// TwinCAT 3 PLC project PLC_MAIN
// ProgramVersion: 3.1.4024.0
// libraries:
//   Tc2_MC2, * (Beckhoff Automation GmbH)
//   Tc2_NC, * (Beckhoff Automation GmbH)
//   Tc2_Standard, * (Beckhoff Automation GmbH)
//   Tc2_System, * (Beckhoff Automation GmbH)
//   Tc2_Utilities, * (Beckhoff Automation GmbH)
//   Tc3_IotBase, * (Beckhoff Automation GmbH)
//   Tc3_JsonXml, * (Beckhoff Automation GmbH)
//   Tc3_Module, * (Beckhoff Automation GmbH)
//   VisuDialogs, * (System)
//   VisuSymbols,3.5.10.0,System
// project tree:
//   DUTs/ E_autoState.TcDUT, E_ECmotorErrorState.TcDUT, E_manualState.TcDUT, E_motorErrorList.TcDUT, E_resetAutoState.TcDUT, E_safetyState.TcDUT, E_teknicMotorMethods.TcDUT, ST_eflexMsgIn.TcDUT, ST_errorRef.TcDUT, ST_ignitionClient.TcDUT
//   / GlobalTextList.TcGTLO, PlcTask.TcTTO, Visualization Manager.TcVMO (not stored), VISU_TASK.TcTTO
//   GVLs/ GVL_devices.TcGVL, GVL_eflex.TcGVL, GVL_ignition.TcGVL, GVL_machine.TcGVL, GVL_persistent.TcGVL
//   POUs/DEVICES/ FB_digitalOut.TcPOU, FB_distSensor2011.TcPOU, FB_estop.TcPOU, FB_ltBar.TcPOU, FB_ltCurtains.TcPOU, FB_pushBtnNC.TcPOU, FB_pushBtnNO.TcPOU, FB_table.TcPOU, FB_teknicMotorEC.TcPOU
//   POUs/FUNCTIONS/ FB_homeToTorque.TcPOU, FB_homeToSensorCustom.TcPOU, FB_ignitionClientHandler.TcPOU, FB_moveToTorque.TcPOU, FB_MultiMotorController.TcPOU, F_checkCoupledMovement.TcPOU, F_checkMoveFinish.TcPOU, F_recordErrorData.TcPOU
//   POUs/ICONS/ Icons.TcIPO (not stored)
//   POUs/LISTS/ actionSelectList.TcTLO
//   POUs/PROGRAMS/ auto.TcPOU, eflex.TcPOU, errorHandling.TcPOU, MAIN.TcPOU, multiControl.TcPOU, manual.TcPOU, motorsInit.TcPOU, tempEflex.TcPOU, updateMotors.TcPOU
//   VISUs/VISUs/Auto Screens/ baseInSkiOutScreen.TcVIS, continueAutoScreen.TcVIS, eflexScreen.TcVIS, loadSpaScreen.TcVIS, machineHomingScreen.TcVIS, studsInScreen.TcVIS, tempEflexScreen.TcVIS, unloadSpaScreen.TcVIS
//   VISUs/VISUs/multiControlScreens/ parametersScreen.TcVIS, multiControlHelp.TcVIS, multiControlScreen.TcVIS, machineMapScreen.TcVIS, motorControlScreen.TcVIS
//   VISUs/VISUs/ errorScreen.TcVIS, mainScreen.TcVIS, manualBypassedScreen.TcVIS, manualScreen.TcVIS, safetyDisableWarning.TcVIS, safetyResetScreen.TcVIS, settingsScreen.TcVIS
// real-time tasks:
//   TASK PlcTask: cycle T#5ms, priority 10, ADS port 350
//   TASK VISU_TASK: cycle T#100000us, priority 12, ADS port 351
// motion (NC):
//   TASK NC-Task 1 SAF: cycle T#1ms, priority 4, ADS port 501
//   TASK NC-Task 1 SVB: cycle T#1ms, priority 6, ADS port 511
//   AXIS LFTROTATION (id 2)
//     General: UnitName=°
//     Dynamic: AccelerationMaximum=55, DecelerationMaximum=55, Acceleration=50, Deceleration=50
//     Velo: RefSearch=3, RefSync=3, SlowManual=5, FastManual=9, Maximum=10
//     OtherSettings: AllowMotionCmdToSlave=true
//     encoder EncType=19
//       EncPara: ScaleFactorNumerator=7.028e-05, MaxCount=#xffffffff
//         SoftEndMinControl: Enable=true, Range=-290
//         SoftEndMaxControl: Enable=true, Range=-65.5
//     drive DrvType=16
//       DrvPara: MaxCount=#xffffffff, DriveControlDWord=#x00020100
//         Analog: VeloReferenz=8, TorqueSetpointScale=10, ScaleFactorActTorque=0.1
//         TimeComp: TaskDelayCycles=1
//     controller CtrType=1
//       CtrPara: PriorControlFactor=1
//         Observer: BandWidth=20
//   AXIS LFTCLAMP (id 1)
//     Dynamic: AccelerationMaximum=105, DecelerationMaximum=105, Acceleration=100, Deceleration=100
//     Velo: RefSearch=20, RefSync=20, SlowManual=20, FastManual=30, Maximum=35
//     OtherSettings: AllowMotionCmdToSlave=true
//     encoder EncType=19
//       EncPara: ScaleFactorNumerator=4.8672e-05, MaxCount=#xffffffff
//         SoftEndMinControl: Enable=true, Range=-260
//         SoftEndMaxControl: Enable=true
//     drive DrvType=16
//       DrvPara: MaxCount=#xffffffff, DriveControlDWord=#x00020100
//         Analog: VeloReferenz=20, TorqueSetpointScale=10, ScaleFactorActTorque=0.1
//         TimeComp: TaskDelayCycles=1
//     controller CtrType=1
//       CtrPara: PriorControlFactor=1
//         Observer: BandWidth=20
//   AXIS Column1 (id 4)
//     Dynamic: AccelerationMaximum=201, DecelerationMaximum=201, Acceleration=200, Deceleration=200
//     Velo: RefSearch=10, RefSync=10, SlowManual=5, FastManual=10, Maximum=15
//     OtherSettings: AllowMotionCmdToSlave=true
//     encoder EncType=19
//       EncPara: ScaleFactorNumerator=9.75e-05, ScaleFactorDenominator=10, MaxCount=#xffffffff
//         SoftEndMinControl: Enable=true, Range=-622
//         SoftEndMaxControl: Range=0.1
//     drive DrvType=16
//       DrvPara: MaxCount=#xffffffff, DriveControlDWord=#x00020100
//         Analog: VeloReferenz=10, TorqueSetpointScale=10, ScaleFactorActTorque=0.1
//         TimeComp: TaskDelayCycles=1
//     controller CtrType=1
//       CtrPara: PriorControlFactor=1
//         Observer: BandWidth=20
//   AXIS LFTWIDTH (id 5)
//     Dynamic: AccelerationMaximum=55, DecelerationMaximum=55, Acceleration=50, Deceleration=50
//     Velo: RefSearch=10, RefSync=10, SlowManual=10, FastManual=20, Maximum=25
//     OtherSettings: AllowMotionCmdToSlave=true
//     encoder EncType=19
//       EncPara: ScaleFactorNumerator=9.7263e-05, MaxCount=#xffffffff
//         SoftEndMinControl: Enable=true
//         SoftEndMaxControl: Enable=true, Range=430
//     drive DrvType=16
//       DrvPara: MaxCount=#xffffffff, DriveControlDWord=#x00020100
//         Analog: VeloReferenz=20, TorqueSetpointScale=10, ScaleFactorActTorque=0.1
//         TimeComp: TaskDelayCycles=1
//     controller CtrType=1
//       CtrPara: PriorControlFactor=1
//         Observer: BandWidth=20
//   AXIS RHTWIDTH (id 6)
//     Dynamic: AccelerationMaximum=55, DecelerationMaximum=55, Acceleration=50, Deceleration=50
//     Velo: RefSearch=10, RefSync=10, SlowManual=20, FastManual=20, Maximum=25
//     OtherSettings: AllowMotionCmdToSlave=true
//     encoder EncType=19
//       EncPara: ScaleFactorNumerator=9.7263e-05, MaxCount=#xffffffff
//         SoftEndMinControl: Enable=true
//         SoftEndMaxControl: Enable=true, Range=430
//     drive DrvType=16
//       DrvPara: MaxCount=#xffffffff, DriveControlDWord=#x00020100
//         Analog: VeloReferenz=20, TorqueSetpointScale=10, ScaleFactorActTorque=0.1
//         TimeComp: TaskDelayCycles=1
//     controller CtrType=1
//       CtrPara: PriorControlFactor=1
//         Observer: BandWidth=20
//   AXIS Column2 (id 7)
//     Dynamic: AccelerationMaximum=201, DecelerationMaximum=201, Acceleration=200, Deceleration=200
//     Velo: RefSearch=10, RefSync=10, Maximum=15
//     OtherSettings: AllowMotionCmdToSlave=true
//     encoder EncType=19
//       EncPara: ScaleFactorNumerator=9.75e-05, ScaleFactorDenominator=10, MaxCount=#xffffffff
//         SoftEndMinControl: Enable=true, Range=-622
//         SoftEndMaxControl: Enable=true
//     drive DrvType=16
//       DrvPara: MaxCount=#xffffffff, DriveControlDWord=#x00020100
//         Analog: VeloReferenz=10, TorqueSetpointScale=10, ScaleFactorActTorque=0.1
//         TimeComp: TaskDelayCycles=1
//     controller CtrType=1
//       CtrPara: PriorControlFactor=1
//         Observer: BandWidth=20
//   AXIS Column3 (id 8)
//     Dynamic: AccelerationMaximum=201, DecelerationMaximum=201, Acceleration=200, Deceleration=200
//     Velo: RefSearch=10, RefSync=10, Maximum=15
//     OtherSettings: AllowMotionCmdToSlave=true
//     encoder EncType=19
//       EncPara: ScaleFactorNumerator=9.75e-05, ScaleFactorDenominator=10, MaxCount=#xffffffff
//         SoftEndMinControl: Enable=true, Range=-622
//         SoftEndMaxControl: Range=0.1
//     drive DrvType=16
//       DrvPara: MaxCount=#xffffffff, DriveControlDWord=#x00020100
//         Analog: VeloReferenz=10, TorqueSetpointScale=10, ScaleFactorActTorque=0.1
//         TimeComp: TaskDelayCycles=1
//     controller CtrType=1
//       CtrPara: PriorControlFactor=1
//         Observer: BandWidth=20
//   AXIS RHTCLAMP (id 9)
//     Dynamic: AccelerationMaximum=105, DecelerationMaximum=105, Acceleration=100, Deceleration=100
//     Velo: RefSearch=20, RefSync=20, SlowManual=20, FastManual=30, Maximum=35
//     OtherSettings: AllowMotionCmdToSlave=true
//     encoder EncType=19
//       EncPara: ScaleFactorNumerator=4.8672e-05, MaxCount=#xffffffff
//         SoftEndMinControl: Enable=true
//         SoftEndMaxControl: Enable=true, Range=260
//     drive DrvType=16
//       DrvPara: MaxCount=#xffffffff, DriveControlDWord=#x00020100
//         Analog: VeloReferenz=20, TorqueSetpointScale=10, ScaleFactorActTorque=0.1
//         TimeComp: TaskDelayCycles=1
//     controller CtrType=1
//       CtrPara: PriorControlFactor=1
//         Observer: BandWidth=20
//   AXIS RHTROTATION (id 10)
//     General: UnitName=°
//     Dynamic: AccelerationMaximum=55, DecelerationMaximum=55, Acceleration=50, Deceleration=50
//     Velo: RefSearch=3, RefSync=3, Maximum=10
//     OtherSettings: AllowMotionCmdToSlave=true
//     encoder EncType=19
//       EncPara: ScaleFactorNumerator=7.028e-05, MaxCount=#xffffffff
//         SoftEndMinControl: Enable=true, Range=67
//         SoftEndMaxControl: Enable=true, Range=290
//     drive DrvType=16
//       DrvPara: MaxCount=#xffffffff, DriveControlDWord=#x00020100
//         Analog: VeloReferenz=8, TorqueSetpointScale=10, ScaleFactorActTorque=0.1
//         TimeComp: TaskDelayCycles=1
//     controller CtrType=1
//       CtrPara: PriorControlFactor=1
//         Observer: BandWidth=20
//   AXIS Column0 (id 11)
//     Dynamic: AccelerationMaximum=201, DecelerationMaximum=201, Acceleration=200, Deceleration=200
//     Velo: RefSearch=10, RefSync=10, SlowManual=10, FastManual=10, Maximum=15
//     OtherSettings: AllowMotionCmdToSlave=true
//     encoder EncType=19
//       EncPara: ScaleFactorNumerator=9.75e-05, ScaleFactorDenominator=10, MaxCount=#xffffffff
//         SoftEndMinControl: Enable=true, Range=-622
//         SoftEndMaxControl: Enable=true
//     drive DrvType=16
//       DrvPara: MaxCount=#xffffffff, DriveControlDWord=#x00020100
//         Analog: VeloReferenz=10, TorqueSetpointScale=10, ScaleFactorActTorque=0.1
//         TimeComp: TaskDelayCycles=1
//     controller CtrType=1
//       CtrPara: PriorControlFactor=1
//         Observer: BandWidth=20
// I/O:
//   DEVICE Device 1 (EtherCAT), AmsNetId 5.151.65.180.2.1
//     Term 10 (EK1200) [EK1200-5000 EtherCAT Power supply (2A E-Bus)]
//       Term 11 (EL1008) [EL1008 8Ch. Dig. Input 24V, 3ms]
//       Term 12 (EL2008) [EL2008 8Ch. Dig. Output 24V, 0.5A]
//       Term 13 (EL2008) [EL2008 8Ch. Dig. Output 24V, 0.5A]
//       Term 14 (EL2904) [EL2904, 4 Ch. Safety Output 24V, 0.5A, TwinSAFE]
//         modules: Module 1 (FSOES), Module 2 (DO)
//       Term 15 (EL3024) [EL3024 4Ch. Ana. Input 4-20mA DIFF]
//       Term 16 (EL3024) [EL3024 4Ch. Ana. Input 4-20mA DIFF]
//       Term 17 (EL1918) [EL1918, 8Ch. Safety Input 24V, TwinSAFE]
//         modules: Module 2 (FSLOGIC)
//       Term 18 (EK1110) [EK1110 EtherCAT extension]
//     Drive 19 (ClearPath EtherCAT Integrated ServoMotor) [ClearPath EC (CoE Rev 2)]
//     Drive 20 (ClearPath EtherCAT Integrated ServoMotor) [ClearPath EC (CoE Rev 2)]
//     Drive 21 (ClearPath EtherCAT Integrated ServoMotor) [ClearPath EC (CoE Rev 2)]
//     Drive 22 (ClearPath EtherCAT Integrated ServoMotor) [ClearPath EC (CoE Rev 2)]
//     Drive 23 (ClearPath EtherCAT Integrated ServoMotor) [ClearPath EC (CoE Rev 2)]
//     Drive 24 (ClearPath EtherCAT Integrated ServoMotor) [ClearPath EC (CoE Rev 2)]
//     Drive 25 (ClearPath EtherCAT Integrated ServoMotor) [ClearPath EC (CoE Rev 2)]
//     Drive 26 (ClearPath EtherCAT Integrated ServoMotor) [ClearPath EC (CoE Rev 2)]
//     Drive 37 (ClearPath EtherCAT Integrated ServoMotor) [ClearPath EC (CoE Rev 2)]
//     Drive 28 (ClearPath EtherCAT Integrated ServoMotor) [ClearPath EC (CoE Rev 2)]
// variable links:
//   PLC_MAIN/PLC_MAIN Instance <-> Device 1 (EtherCAT)/Term 10 (EK1200)/Term 11 (EL1008)
//     PlcTask Inputs/GVL_devices.fbColumn0Motor.bHomeSensor <-> Channel 6/Input
//     PlcTask Inputs/GVL_devices.fbColumn2Motor.bHomeSensor <-> Channel 5/Input
//     PlcTask Inputs/GVL_devices.fbLftWidthMotor.bClampSensor <-> Channel 1/Input
//     PlcTask Inputs/GVL_devices.fbLftWidthMotor.bHomeSensor <-> Channel 4/Input
//     PlcTask Inputs/GVL_devices.fbRhtWidthMotor.bClampSensor <-> Channel 2/Input
//     PlcTask Inputs/GVL_devices.fbRhtWidthMotor.bHomeSensor <-> Channel 3/Input
//     PlcTask Inputs/GVL_devices.fbTable.bLoadedSensor <-> Channel 7/Input
//   PLC_MAIN/PLC_MAIN Instance <-> Device 1 (EtherCAT)/Term 10 (EK1200)/Term 12 (EL2008)
//     PlcTask Outputs/GVL_devices.fbLftClampMotor.bBrake <-> Channel 7/Output
//     PlcTask Outputs/GVL_devices.fbLftRotationMotor.bBrake <-> Channel 4/Output
//     PlcTask Outputs/GVL_devices.fbLtBars.bGreenLight <-> Channel 1/Output
//     PlcTask Outputs/GVL_devices.fbLtBars.bRedLight <-> Channel 3/Output
//     PlcTask Outputs/GVL_devices.fbLtBars.bYellowLight <-> Channel 2/Output
//     PlcTask Outputs/GVL_devices.fbRhtClampMotor.bBrake <-> Channel 6/Output
//     PlcTask Outputs/GVL_devices.fbRhtRotationMotor.bBrake <-> Channel 5/Output
//   PLC_MAIN/PLC_MAIN Instance <-> Device 1 (EtherCAT)/Term 10 (EK1200)/Term 13 (EL2008)
//     PlcTask Outputs/GVL_devices.fbTable.bTableBlackWire <-> Channel 5/Output
//     PlcTask Outputs/GVL_devices.fbTable.bTableBlueWire <-> Channel 6/Output
//     PlcTask Outputs/GVL_devices.fbTable.bTableGreenWire <-> Channel 4/Output
//   PLC_MAIN/PLC_MAIN Instance <-> Device 1 (EtherCAT)/Term 10 (EK1200)/Term 16 (EL3024)
//     PlcTask Inputs/GVL_devices.fbTable.tableDistSens.nSensor <-> AI Standard Channel 1/Value
//   PLC_MAIN/PLC_MAIN Instance <-> Device 1 (EtherCAT)/Term 10 (EK1200)/Term 17 (EL1918)
//     PlcTask Inputs/GVL_devices.fbEstop.bEstopFbError <-> StandardInputs/Standard Out Var 18
//     PlcTask Inputs/GVL_devices.fbEstop.bEstopSigOk <-> StandardInputs/Standard Out Var 19
//     PlcTask Inputs/GVL_devices.fbEstop.nEstopFbState <-> Function Block Info Data/TwinSafeGroup1.Network1.FBEstop1 Info Data/State
//     PlcTask Inputs/GVL_devices.fbLtCurtains.bCurtainsMuted <-> StandardInputs/Standard Out Var 17
//     PlcTask Inputs/GVL_devices.fbLtCurtains.bLftCurtainFbError <-> StandardInputs/Standard Out Var 11
//     PlcTask Inputs/GVL_devices.fbLtCurtains.bLftCurtainSigOk <-> StandardInputs/Standard Out Var 12
//     PlcTask Inputs/GVL_devices.fbLtCurtains.bRhtCurtainFbError <-> StandardInputs/Standard Out Var 14
//     PlcTask Inputs/GVL_devices.fbLtCurtains.bRhtCurtainSigOk <-> StandardInputs/Standard Out Var 15
//     PlcTask Inputs/GVL_devices.fbLtCurtains.nLftCurtainFbState <-> Function Block Info Data/TwinSafeGroup1.Network1.FBMon1 Info Data/State
//     PlcTask Inputs/GVL_devices.fbLtCurtains.nRhtCurtainFbState <-> Function Block Info Data/TwinSafeGroup1.Network1.FBMon2 Info Data/State
//     PlcTask Inputs/GVL_machine.bComErr <-> StandardInputs/Standard Out Var 8
//     PlcTask Inputs/GVL_machine.bFbErr <-> StandardInputs/Standard Out Var 20
//     PlcTask Inputs/GVL_machine.bFbRun <-> StandardInputs/Standard Out Var 9
//     PlcTask Inputs/GVL_machine.bInRun <-> StandardInputs/Standard Out Var 10
//     PlcTask Inputs/GVL_machine.bOtherErr <-> StandardInputs/Standard Out Var 13
//     PlcTask Inputs/GVL_machine.bSafetyOk <-> StandardInputs/Standard Out Var 16
//     PlcTask Outputs/GVL_devices.fbEstop.bResetEstopFb <-> StandardOutputs/Standard In Var 4
//     PlcTask Outputs/GVL_devices.fbLtCurtains.bMuteCurtains <-> StandardOutputs/Standard In Var 3
//     PlcTask Outputs/GVL_devices.fbLtCurtains.bResetLftCurtainFb <-> StandardOutputs/Standard In Var 5
//     PlcTask Outputs/GVL_devices.fbLtCurtains.bResetRhtCurtainFb <-> StandardOutputs/Standard In Var 6
//     PlcTask Outputs/GVL_machine.bRunSafety <-> StandardOutputs/Standard In Var 2
//     PlcTask Outputs/GVL_machine.bSafetyBypass <-> StandardOutputs/Standard In Var 7
//     PlcTask Outputs/GVL_machine.bSafetyErrorAck <-> StandardOutputs/Standard In Var 1
//   PLC_MAIN/PLC_MAIN Instance <-> NC-Task 1 SAF/Axes/Column0
//     PlcTask Inputs/GVL_devices.fbColumn0Motor.fbMotor.NcToPlc <-> Outputs/ToPlc
//     PlcTask Outputs/GVL_devices.fbColumn0Motor.fbMotor.PlcToNc <-> Inputs/FromPlc
//   PLC_MAIN/PLC_MAIN Instance <-> NC-Task 1 SAF/Axes/Column1
//     PlcTask Inputs/GVL_devices.fbColumn1Motor.fbMotor.NcToPlc <-> Outputs/ToPlc
//     PlcTask Outputs/GVL_devices.fbColumn1Motor.fbMotor.PlcToNc <-> Inputs/FromPlc
//   PLC_MAIN/PLC_MAIN Instance <-> NC-Task 1 SAF/Axes/Column2
//     PlcTask Inputs/GVL_devices.fbColumn2Motor.fbMotor.NcToPlc <-> Outputs/ToPlc
//     PlcTask Outputs/GVL_devices.fbColumn2Motor.fbMotor.PlcToNc <-> Inputs/FromPlc
//   PLC_MAIN/PLC_MAIN Instance <-> NC-Task 1 SAF/Axes/Column3
//     PlcTask Inputs/GVL_devices.fbColumn3Motor.fbMotor.NcToPlc <-> Outputs/ToPlc
//     PlcTask Outputs/GVL_devices.fbColumn3Motor.fbMotor.PlcToNc <-> Inputs/FromPlc
//   PLC_MAIN/PLC_MAIN Instance <-> NC-Task 1 SAF/Axes/LFTCLAMP
//     PlcTask Inputs/GVL_devices.fbLftClampMotor.fbMotor.NcToPlc <-> Outputs/ToPlc
//     PlcTask Outputs/GVL_devices.fbLftClampMotor.fbMotor.PlcToNc <-> Inputs/FromPlc
//   PLC_MAIN/PLC_MAIN Instance <-> NC-Task 1 SAF/Axes/LFTROTATION
//     PlcTask Inputs/GVL_devices.fbLftRotationMotor.fbMotor.NcToPlc <-> Outputs/ToPlc
//     PlcTask Outputs/GVL_devices.fbLftRotationMotor.fbMotor.PlcToNc <-> Inputs/FromPlc
//   PLC_MAIN/PLC_MAIN Instance <-> NC-Task 1 SAF/Axes/LFTWIDTH
//     PlcTask Inputs/GVL_devices.fbLftWidthMotor.fbMotor.NcToPlc <-> Outputs/ToPlc
//     PlcTask Outputs/GVL_devices.fbLftWidthMotor.fbMotor.PlcToNc <-> Inputs/FromPlc
//   PLC_MAIN/PLC_MAIN Instance <-> NC-Task 1 SAF/Axes/RHTCLAMP
//     PlcTask Inputs/GVL_devices.fbRhtClampMotor.fbMotor.NcToPlc <-> Outputs/ToPlc
//     PlcTask Outputs/GVL_devices.fbRhtClampMotor.fbMotor.PlcToNc <-> Inputs/FromPlc
//   PLC_MAIN/PLC_MAIN Instance <-> NC-Task 1 SAF/Axes/RHTROTATION
//     PlcTask Inputs/GVL_devices.fbRhtRotationMotor.fbMotor.NcToPlc <-> Outputs/ToPlc
//     PlcTask Outputs/GVL_devices.fbRhtRotationMotor.fbMotor.PlcToNc <-> Inputs/FromPlc
//   PLC_MAIN/PLC_MAIN Instance <-> NC-Task 1 SAF/Axes/RHTWIDTH
//     PlcTask Inputs/GVL_devices.fbRhtWidthMotor.fbMotor.NcToPlc <-> Outputs/ToPlc
//     PlcTask Outputs/GVL_devices.fbRhtWidthMotor.fbMotor.PlcToNc <-> Inputs/FromPlc
//   Axes/LFTROTATION <-> Device 1 (EtherCAT)/Drive 19 (ClearPath EtherCAT Integrated ServoMotor)
//     Drive/Inputs/In/nDataIn1 <-> TxPDO 1/Following Error Actual Value
//     Drive/Inputs/In/nDataIn3[0] <-> TxPDO 1/Torque Actual Value
//     Drive/Inputs/In/nState1 <-> TxPDO 1/Statusword
//     Drive/Inputs/In/nState2 <-> TxPDO 1/Statusword @bit 8
//     Drive/Inputs/In/nState4 @bit 1 <-> WcState/InputToggle
//     Drive/Inputs/In/nState4 <-> WcState/WcState
//     Drive/Inputs/In/nState5 <-> TxPDO 1/Modes of Operation Display
//     Drive/Outputs/Out/nCtrl1 <-> RxPDO 1/Controlword
//     Drive/Outputs/Out/nCtrl2 <-> RxPDO 1/Controlword @bit 8
//     Drive/Outputs/Out/nCtrl5 <-> RxPDO 1/Modes of Operation
//     Drive/Outputs/Out/nDataOut1 <-> RxPDO 1/Target Position
//     Drive/Outputs/Out/nDataOut2 <-> RxPDO 1/Target Velocity
//     Drive/Outputs/Out/nDataOut4[0] <-> RxPDO 1/Target Torque
//     Enc/Inputs/In/nDataIn1 <-> TxPDO 1/Position Actual Value
//     Enc/Inputs/In/nDataIn7 <-> TxPDO 1/Velocity Actual Value
//     Enc/Inputs/In/nState4 @bit 1 <-> WcState/InputToggle
//     Enc/Inputs/In/nState4 <-> WcState/WcState
//   (this object) <-> Device 1 (EtherCAT)/Drive 20 (ClearPath EtherCAT Integrated ServoMotor)
//     Drive/Inputs/In/nDataIn1 <-> TxPDO 1/Following Error Actual Value
//     Drive/Inputs/In/nDataIn3[0] <-> TxPDO 1/Torque Actual Value
//     Drive/Inputs/In/nState1 <-> TxPDO 1/Statusword
//     Drive/Inputs/In/nState2 <-> TxPDO 1/Statusword @bit 8
//     Drive/Inputs/In/nState4 @bit 1 <-> WcState/InputToggle
//     Drive/Inputs/In/nState4 <-> WcState/WcState
//     Drive/Inputs/In/nState5 <-> TxPDO 1/Modes of Operation Display
//     Drive/Outputs/Out/nCtrl1 <-> RxPDO 1/Controlword
//     Drive/Outputs/Out/nCtrl2 <-> RxPDO 1/Controlword @bit 8
//     Drive/Outputs/Out/nCtrl5 <-> RxPDO 1/Modes of Operation
//     Drive/Outputs/Out/nDataOut1 <-> RxPDO 1/Target Position
//     Drive/Outputs/Out/nDataOut2 <-> RxPDO 1/Target Velocity
//     Drive/Outputs/Out/nDataOut4[0] <-> RxPDO 1/Target Torque
//     Enc/Inputs/In/nDataIn1 <-> TxPDO 1/Position Actual Value
//     Enc/Inputs/In/nDataIn7 <-> TxPDO 1/Velocity Actual Value
//     Enc/Inputs/In/nState4 @bit 1 <-> WcState/InputToggle
//     Enc/Inputs/In/nState4 <-> WcState/WcState
//   (this object) <-> Device 1 (EtherCAT)/Drive 22 (ClearPath EtherCAT Integrated ServoMotor)
//     Drive/Inputs/In/nDataIn1 <-> TxPDO 1/Following Error Actual Value
//     Drive/Inputs/In/nDataIn3[0] <-> TxPDO 1/Torque Actual Value
//     Drive/Inputs/In/nState1 <-> TxPDO 1/Statusword
//     Drive/Inputs/In/nState2 <-> TxPDO 1/Statusword @bit 8
//     Drive/Inputs/In/nState4 @bit 1 <-> WcState/InputToggle
//     Drive/Inputs/In/nState4 <-> WcState/WcState
//     Drive/Inputs/In/nState5 <-> TxPDO 1/Modes of Operation Display
//     Drive/Outputs/Out/nCtrl1 <-> RxPDO 1/Controlword
//     Drive/Outputs/Out/nCtrl2 <-> RxPDO 1/Controlword @bit 8
//     Drive/Outputs/Out/nCtrl5 <-> RxPDO 1/Modes of Operation
//     Drive/Outputs/Out/nDataOut1 <-> RxPDO 1/Target Position
//     Drive/Outputs/Out/nDataOut2 <-> RxPDO 1/Target Velocity
//     Drive/Outputs/Out/nDataOut4[0] <-> RxPDO 1/Target Torque
//     Enc/Inputs/In/nDataIn1 <-> TxPDO 1/Position Actual Value
//     Enc/Inputs/In/nDataIn7 <-> TxPDO 1/Velocity Actual Value
//     Enc/Inputs/In/nState4 @bit 1 <-> WcState/InputToggle
//     Enc/Inputs/In/nState4 <-> WcState/WcState
//   (this object) <-> Device 1 (EtherCAT)/Drive 23 (ClearPath EtherCAT Integrated ServoMotor)
//     Drive/Inputs/In/nDataIn1 <-> TxPDO 1/Following Error Actual Value
//     Drive/Inputs/In/nDataIn3[0] <-> TxPDO 1/Torque Actual Value
//     Drive/Inputs/In/nState1 <-> TxPDO 1/Statusword
//     Drive/Inputs/In/nState2 <-> TxPDO 1/Statusword @bit 8
//     Drive/Inputs/In/nState4 @bit 1 <-> WcState/InputToggle
//     Drive/Inputs/In/nState4 <-> WcState/WcState
//     Drive/Inputs/In/nState5 <-> TxPDO 1/Modes of Operation Display
//     Drive/Outputs/Out/nCtrl1 <-> RxPDO 1/Controlword
//     Drive/Outputs/Out/nCtrl2 <-> RxPDO 1/Controlword @bit 8
//     Drive/Outputs/Out/nCtrl5 <-> RxPDO 1/Modes of Operation
//     Drive/Outputs/Out/nDataOut1 <-> RxPDO 1/Target Position
//     Drive/Outputs/Out/nDataOut2 <-> RxPDO 1/Target Velocity
//     Drive/Outputs/Out/nDataOut4[0] <-> RxPDO 1/Target Torque
//     Enc/Inputs/In/nDataIn1 <-> TxPDO 1/Position Actual Value
//     Enc/Inputs/In/nDataIn7 <-> TxPDO 1/Velocity Actual Value
//     Enc/Inputs/In/nState4 @bit 1 <-> WcState/InputToggle
//     Enc/Inputs/In/nState4 <-> WcState/WcState
//   (this object) <-> Device 1 (EtherCAT)/Drive 24 (ClearPath EtherCAT Integrated ServoMotor)
//     Drive/Inputs/In/nDataIn1 <-> TxPDO 1/Following Error Actual Value
//     Drive/Inputs/In/nDataIn3[0] <-> TxPDO 1/Torque Actual Value
//     Drive/Inputs/In/nState1 <-> TxPDO 1/Statusword
//     Drive/Inputs/In/nState2 <-> TxPDO 1/Statusword @bit 8
//     Drive/Inputs/In/nState4 @bit 1 <-> WcState/InputToggle
//     Drive/Inputs/In/nState4 <-> WcState/WcState
//     Drive/Inputs/In/nState5 <-> TxPDO 1/Modes of Operation Display
//     Drive/Outputs/Out/nCtrl1 <-> RxPDO 1/Controlword
//     Drive/Outputs/Out/nCtrl2 <-> RxPDO 1/Controlword @bit 8
//     Drive/Outputs/Out/nCtrl5 <-> RxPDO 1/Modes of Operation
//     Drive/Outputs/Out/nDataOut1 <-> RxPDO 1/Target Position
//     Drive/Outputs/Out/nDataOut2 <-> RxPDO 1/Target Velocity
//     Drive/Outputs/Out/nDataOut4[0] <-> RxPDO 1/Target Torque
//     Enc/Inputs/In/nDataIn1 <-> TxPDO 1/Position Actual Value
//     Enc/Inputs/In/nDataIn7 <-> TxPDO 1/Velocity Actual Value
//     Enc/Inputs/In/nState4 @bit 1 <-> WcState/InputToggle
//     Enc/Inputs/In/nState4 <-> WcState/WcState
//   (this object) <-> Device 1 (EtherCAT)/Drive 25 (ClearPath EtherCAT Integrated ServoMotor)
//     Drive/Inputs/In/nDataIn1 <-> TxPDO 1/Following Error Actual Value
//     Drive/Inputs/In/nDataIn3[0] <-> TxPDO 1/Torque Actual Value
//     Drive/Inputs/In/nState1 <-> TxPDO 1/Statusword
//     Drive/Inputs/In/nState2 <-> TxPDO 1/Statusword @bit 8
//     Drive/Inputs/In/nState4 @bit 1 <-> WcState/InputToggle
//     Drive/Inputs/In/nState4 <-> WcState/WcState
//     Drive/Inputs/In/nState5 <-> TxPDO 1/Modes of Operation Display
//     Drive/Outputs/Out/nCtrl1 <-> RxPDO 1/Controlword
//     Drive/Outputs/Out/nCtrl2 <-> RxPDO 1/Controlword @bit 8
//     Drive/Outputs/Out/nCtrl5 <-> RxPDO 1/Modes of Operation
//     Drive/Outputs/Out/nDataOut1 <-> RxPDO 1/Target Position
//     Drive/Outputs/Out/nDataOut2 <-> RxPDO 1/Target Velocity
//     Drive/Outputs/Out/nDataOut4[0] <-> RxPDO 1/Target Torque
//     Enc/Inputs/In/nDataIn1 <-> TxPDO 1/Position Actual Value
//     Enc/Inputs/In/nDataIn7 <-> TxPDO 1/Velocity Actual Value
//     Enc/Inputs/In/nState4 @bit 1 <-> WcState/InputToggle
//     Enc/Inputs/In/nState4 <-> WcState/WcState
//   (this object) <-> Device 1 (EtherCAT)/Drive 26 (ClearPath EtherCAT Integrated ServoMotor)
//     Drive/Inputs/In/nDataIn1 <-> TxPDO 1/Following Error Actual Value
//     Drive/Inputs/In/nDataIn3[0] <-> TxPDO 1/Torque Actual Value
//     Drive/Inputs/In/nState1 <-> TxPDO 1/Statusword
//     Drive/Inputs/In/nState2 <-> TxPDO 1/Statusword @bit 8
//     Drive/Inputs/In/nState4 @bit 1 <-> WcState/InputToggle
//     Drive/Inputs/In/nState4 <-> WcState/WcState
//     Drive/Inputs/In/nState5 <-> TxPDO 1/Modes of Operation Display
//     Drive/Outputs/Out/nCtrl1 <-> RxPDO 1/Controlword
//     Drive/Outputs/Out/nCtrl2 <-> RxPDO 1/Controlword @bit 8
//     Drive/Outputs/Out/nCtrl5 <-> RxPDO 1/Modes of Operation
//     Drive/Outputs/Out/nDataOut1 <-> RxPDO 1/Target Position
//     Drive/Outputs/Out/nDataOut2 <-> RxPDO 1/Target Velocity
//     Drive/Outputs/Out/nDataOut4[0] <-> RxPDO 1/Target Torque
//     Enc/Inputs/In/nDataIn1 <-> TxPDO 1/Position Actual Value
//     Enc/Inputs/In/nDataIn7 <-> TxPDO 1/Velocity Actual Value
//     Enc/Inputs/In/nState4 @bit 1 <-> WcState/InputToggle
//     Enc/Inputs/In/nState4 <-> WcState/WcState
//   (this object) <-> Device 1 (EtherCAT)/Drive 37 (ClearPath EtherCAT Integrated ServoMotor)
//     Drive/Inputs/In/nDataIn1 <-> TxPDO 1/Following Error Actual Value
//     Drive/Inputs/In/nDataIn3[0] <-> TxPDO 1/Torque Actual Value
//     Drive/Inputs/In/nState1 <-> TxPDO 1/Statusword
//     Drive/Inputs/In/nState2 <-> TxPDO 1/Statusword @bit 8
//     Drive/Inputs/In/nState4 @bit 1 <-> WcState/InputToggle
//     Drive/Inputs/In/nState4 <-> WcState/WcState
//     Drive/Inputs/In/nState5 <-> TxPDO 1/Modes of Operation Display
//     Drive/Outputs/Out/nCtrl1 <-> RxPDO 1/Controlword
//     Drive/Outputs/Out/nCtrl2 <-> RxPDO 1/Controlword @bit 8
//     Drive/Outputs/Out/nCtrl5 <-> RxPDO 1/Modes of Operation
//     Drive/Outputs/Out/nDataOut1 <-> RxPDO 1/Target Position
//     Drive/Outputs/Out/nDataOut2 <-> RxPDO 1/Target Velocity
//     Drive/Outputs/Out/nDataOut4[0] <-> RxPDO 1/Target Torque
//     Enc/Inputs/In/nDataIn1 <-> TxPDO 1/Position Actual Value
//     Enc/Inputs/In/nDataIn7 <-> TxPDO 1/Velocity Actual Value
//     Enc/Inputs/In/nState4 @bit 1 <-> WcState/InputToggle
//     Enc/Inputs/In/nState4 <-> WcState/WcState
//   (this object) <-> Device 1 (EtherCAT)/Drive 28 (ClearPath EtherCAT Integrated ServoMotor)
//     Drive/Inputs/In/nDataIn1 <-> TxPDO 1/Following Error Actual Value
//     Drive/Inputs/In/nDataIn3[0] <-> TxPDO 1/Torque Actual Value
//     Drive/Inputs/In/nState1 <-> TxPDO 1/Statusword
//     Drive/Inputs/In/nState2 <-> TxPDO 1/Statusword @bit 8
//     Drive/Inputs/In/nState4 @bit 1 <-> WcState/InputToggle
//     Drive/Inputs/In/nState4 <-> WcState/WcState
//     Drive/Inputs/In/nState5 <-> TxPDO 1/Modes of Operation Display
//     Drive/Outputs/Out/nCtrl1 <-> RxPDO 1/Controlword
//     Drive/Outputs/Out/nCtrl2 <-> RxPDO 1/Controlword @bit 8
//     Drive/Outputs/Out/nCtrl5 <-> RxPDO 1/Modes of Operation
//     Drive/Outputs/Out/nDataOut1 <-> RxPDO 1/Target Position
//     Drive/Outputs/Out/nDataOut2 <-> RxPDO 1/Target Velocity
//     Drive/Outputs/Out/nDataOut4[0] <-> RxPDO 1/Target Torque
//     Enc/Inputs/In/nDataIn1 <-> TxPDO 1/Position Actual Value
//     Enc/Inputs/In/nDataIn7 <-> TxPDO 1/Velocity Actual Value
//     Enc/Inputs/In/nState4 @bit 1 <-> WcState/InputToggle
//     Enc/Inputs/In/nState4 <-> WcState/WcState
//   (this object) <-> Device 1 (EtherCAT)/Drive 21 (ClearPath EtherCAT Integrated ServoMotor)
//     Drive/Inputs/In/nDataIn1 <-> TxPDO 1/Following Error Actual Value
//     Drive/Inputs/In/nDataIn3[0] <-> TxPDO 1/Torque Actual Value
//     Drive/Inputs/In/nState1 <-> TxPDO 1/Statusword
//     Drive/Inputs/In/nState2 <-> TxPDO 1/Statusword @bit 8
//     Drive/Inputs/In/nState4 @bit 1 <-> WcState/InputToggle
//     Drive/Inputs/In/nState4 <-> WcState/WcState
//     Drive/Inputs/In/nState5 <-> TxPDO 1/Modes of Operation Display
//     Drive/Outputs/Out/nCtrl1 <-> RxPDO 1/Controlword
//     Drive/Outputs/Out/nCtrl2 <-> RxPDO 1/Controlword @bit 8
//     Drive/Outputs/Out/nCtrl5 <-> RxPDO 1/Modes of Operation
//     Drive/Outputs/Out/nDataOut1 <-> RxPDO 1/Target Position
//     Drive/Outputs/Out/nDataOut2 <-> RxPDO 1/Target Velocity
//     Drive/Outputs/Out/nDataOut4[0] <-> RxPDO 1/Target Torque
//     Enc/Inputs/In/nDataIn1 <-> TxPDO 1/Position Actual Value
//     Enc/Inputs/In/nDataIn7 <-> TxPDO 1/Velocity Actual Value
//     Enc/Inputs/In/nState4 @bit 1 <-> WcState/InputToggle
//     Enc/Inputs/In/nState4 <-> WcState/WcState
//   (this object) <-> Device 1 (EtherCAT)
//     Term 10 (EK1200)/Term 14 (EL2904)/Module 1 (FSOES)/RxPDO/FSOE <-> Term 10 (EK1200)/Term 17 (EL1918)/ConnectionInputs/Message_21 TxPDO
//     Term 10 (EK1200)/Term 14 (EL2904)/Module 1 (FSOES)/TxPDO/FSOE <-> Term 10 (EK1200)/Term 17 (EL1918)/ConnectionOutputs/Message_21 RxPDO
//     Term 10 (EK1200)/Term 17 (EL1918)/ConnectionInputs/Message_21 TxPDO <-> Term 10 (EK1200)/Term 14 (EL2904)/Module 1 (FSOES)/RxPDO/FSOE
//     Term 10 (EK1200)/Term 17 (EL1918)/ConnectionOutputs/Message_21 RxPDO <-> Term 10 (EK1200)/Term 14 (EL2904)/Module 1 (FSOES)/TxPDO/FSOE

CONFIGURATION PLC_MAIN
    RESOURCE PLC ON TwinCAT3
        TASK PlcTask(INTERVAL := T#5ms, PRIORITY := 10);
        TASK VISU_TASK(INTERVAL := T#200000us, PRIORITY := 14);
        PROGRAM MAIN WITH PlcTask : MAIN;
        PROGRAM VisuElems_Visu_Prg WITH VISU_TASK : VisuElems.Visu_Prg;
    END_RESOURCE
END_CONFIGURATION

// ---- DUTs/E_autoState.TcDUT
TYPE E_autoState :
(
	CONFIRMINITHOMING := 0,
	INITHOMING,
	SCANEFLEX,
	CONFIRMPROGRAM,
	CONFIRMSTART,
	TABLETOCONVEYOR,
	CONFIRMLOADED,
	TABLETOCLAMP,
	CENTERSPA,
	OPENCLAMP,
	MOVETOCLAMP,
	CLAMPSPA,
	ROTATESPA,
	TABLETOBASE,
	CONFIRMSKIIS,
	CONFIRMBASE,
	LOWERSPA,
	UNCLAMPSPA,
	CLAMPRETURN,
	CONFIRMSPAUNLOAD,
	EXITHOMING,
	INITSTATE,
	RESETPROGRAM,
	STOPPROGRAM,
	RESETMOTORS,
	MOTORFAULTED,
	PROGERRORSTOP,
	RESETLFTCOLUMNS,
	RESETRHTCOLUMNS,
	MATCHLFTCOLUMNS,
	MATCHRHTCOLUMNS,
	CONFIRMMANUALCLAMPING
)DINT;
END_TYPE

// ---- DUTs/E_ECmotorErrorState.TcDUT
TYPE E_ECmotorErrorState :
(
	MCHOME := 0,
	MCREADDRIVEOPERATIONMODE,
	MCWRITEDRIVEOPERATIONMODE,
	MCHALT,
	MCSTOP,
	MCJOG,
	MCMOVEABSOLUTE,
	MCMOVERELATIVE,
	MCPOWER,
	MCRESET,
	MCSETPOSITION,
	MCWRITEPARAMETER,
	MCREADSTATUS,
	MCTORQUECONTROL,
	MCGEARIN,
	MCGEAROUT
)INT;
END_TYPE

// ---- DUTs/E_manualState.TcDUT
TYPE E_manualState :
(
	STEADYSTATE := 0,
	MOVEAWAYDIRECTION,
	MOVEHOMEDIRECTION,
	RESET,
	HOMING
)DINT;
END_TYPE

// ---- DUTs/E_motorErrorList.TcDUT
TYPE E_motorErrorList :
(
	LFTROTATION := 0,
	LFTCLAMP,
	COLUMN0,
	COLUMN1,
	LFTWIDTH,
	RHTWIDTH,
	COLUMN2,
	COLUMN3,
	RHTCLAMP,
	RHTROTATION,
	CUSTOM
)DINT;
END_TYPE

// ---- DUTs/E_resetAutoState.TcDUT
TYPE E_resetAutoState :
(
	CHECKWIDTH := 0,
	CHECKCLAMPS,
	CHECKROTATION,
	CHECKHEIGHT,
	MOVETOFLIPHEIGHT,
	MOVETOUNCLAMPHEIGHT,
	OPENCLAMPS,
	RESETDONE
	
);
END_TYPE

// ---- DUTs/E_safetyState.TcDUT
TYPE E_safetyState :
(
	INIT := 0,
	PREOP,
	OK,
	FAULT,
	WAITRESET,
	RESETTING,
	BYPASS,
	LOCKOUT,
	RESETCURTAINS,
	RESETESTOP,
	ENGAGED
)DINT;
END_TYPE

// ---- DUTs/E_teknicMotorMethods.TcDUT
TYPE E_teknicMotorMethods :
(
	brakeOff := 0,
	brakeOn,
	checkOutputs,
	coupleToAxis,
	decoupleAxis,
	disable,
	enable,
	estop,
	homeToSensor,
	homeToTorque,
	motorInit,
	moveTo,
	moveToJog,
	moveToSensor,
	moveToTorque,
	readMotorParameter,
	removeStop,
	motorReset,
	resetMotorCommands,
	setError,
	stop,
	writeMotorParameter
);
END_TYPE

// ---- DUTs/ST_eflexMsgIn.TcDUT
TYPE ST_eflexMsgIn :
STRUCT
	serialNumber		: STRING;
	taskType			: STRING;
	taskConfigId		: STRING;
	liveBuildStatusId 	: STRING;
	spaModel 			: STRING;
	flipHeight 			: REAL;
	studHeight 			: REAL;
	baseInHeight		: REAL;
	spaOutHeight		: REAL;
END_STRUCT
END_TYPE

// ---- DUTs/ST_errorRef.TcDUT
TYPE ST_errorRef :
STRUCT
	///		errorLoc: Location of the error. i.e. Right Height Motor
	errorLoc : STRING;

	///		errorId: If error is an axis error, the errorId will correlate to axis errors
	///				 found in infoSys
	errorId : UDINT;
	
	///		errorMsg : String representation if any. 'NULL' represents no msg. 'Not Found' represents lookup needed. 
	errorMsg : STRING;
	
	//		errorState: What function block did the error originate from. 
	errorState : E_ECmotorErrorState;
END_STRUCT
END_TYPE

// ---- DUTs/ST_ignitionClient.TcDUT
TYPE ST_ignitionClient :
STRUCT
	sSessionId : STRING;
	sRole : STRING;
	bActive : BOOL;
	bHasControl : BOOL;
END_STRUCT
END_TYPE

// ---- GVLs/GVL_devices.TcGVL
	{attribute 'qualified_only'}
VAR_GLOBAL
	fbLtBars 			: FB_ltBar;
	fbLtCurtains		: FB_ltCurtains;
	fbEstop				: FB_estop;
	fbTable 			: FB_table;
	safetyBuzzer        AT %Q* : BOOL;
	
	fbLftWidthMotor 	: FB_teknicMotorEC;
	fbRhtWidthMotor 	: FB_teknicMotorEC;
	
	fbLftClampMotor 	: FB_teknicMotorEC;
	fbRhtClampMotor 	: FB_teknicMotorEC;
	
	fbLftRotationMotor 	: FB_teknicMotorEC;
	fbRhtRotationMotor 	: FB_teknicMotorEC;
	
	fbColumn0Motor 		: FB_teknicMotorEC;
	fbColumn1Motor 		: FB_teknicMotorEC;
	fbColumn2Motor 		: FB_teknicMotorEC;
	fbColumn3Motor 		: FB_teknicMotorEC;
	
	
END_VAR

// ---- GVLs/GVL_eflex.TcGVL
{attribute 'qualified_only'}
VAR_GLOBAL
	{attribute 'OPC.UA.DA' := '1'}
	bEflexPresent 	: BOOL := FALSE;
	sSpaModel		: STRING;
	fStudHeight		: REAL; // Column Height to lower spa onto base
	fFlipHeight		: REAL; // Column Height to flip spa at
	fBaseInHeight	: REAL; // Table height for recieving base
	fSpaOutHeight	: REAL; //Table height for unloading spa
	
END_VAR

// ---- GVLs/GVL_ignition.TcGVL
{attribute 'qualified_only'}
VAR_GLOBAL
	fTableHeight : REAL;
	fColumnHeight : REAL;
	fClampHeight : REAL;
	fWidthDistance : REAL;
	fRotationDistance : REAL;
	
	
	//Client Handling 
	aIgnitionClients : ARRAY[0..10] OF ST_ignitionClient;
	nNumClients : INT;
	sMachineHMISessionID : STRING(64);
	bControlAssigned : BOOL := FALSE;
	sReqID : STRING;
	sRole : STRING;
	SRemoveID : STRING;
	bClientAddError : BOOL;
	
	//Client Control Request
	sOwnerSessionID 	: STRING(64); // Current controller
	sPendingSessionID	: STRING(64); // Session requesting 
	sRequestedMode		: STRING; //Mode requested to change to
	bTransferRequested 	: BOOL;
	bTransferApproved 	: BOOL;
	bTransferComplete 	: BOOL;
	
	sDenyReason		: STRING(64);
END_VAR

// ---- GVLs/GVL_machine.TcGVL
{attribute 'qualified_only'}
VAR_GLOBAL
	bMotorsInitialized : BOOL;
	sMotorInitState : STRING;
	bPageChange : BOOL;
	bLftColumnsLatched : BOOL;
	bRhtColumnsLatched : BOOL;
	
	///////////////////// SAFETY /////////////////////////////////
	bRunSafety			AT %Q* : BOOL := TRUE; 	// Used to run safety program
	bSafetyErrorAck 	AT %Q* : BOOL; 			// Sequence to acknowledge safety error : False > True > False.
	bSafetyBypass		AT %Q* : BOOL;			//Used to Bypass entire safety PLC. Should Only be accessible with high level credentials. 
	bSafetyOk 			AT %I* : BOOL;			// Safety protocol enacted 
	bFbRun 				AT %I* : BOOL;			// Safety Function Blocks are running
	bInRun				AT %I* : BOOL;			// Safety Program is Running
	bFbErr				AT %I* : BOOL;			// A Safety Function Block contains an error
	bComErr				AT %I* : BOOL;			// Safety program communication error
	bOtherErr			AT %I* : BOOL;			// Other safety error exist. (EDM FB)
	bTestErr			AT %I* : BOOL;
	
	bSafetyInit : BOOL;
	nPageIndex: INT;
	nPrevPageIndex: INT;
	bMotorInitFailedDisp: BOOL;
	bMuteSafety: BOOL;
	
	////////////////////////ERROR HANDLING//////////////////////
	motorErrorList	: E_motorErrorList;
	bErrorPresent 	: BOOL;
	bDispErrorIcon 	: BOOL;
	
	///////////////////////SETTINGS SCREEN//////////////////////
	sEditMessage	: STRING(1024) := 'Changing this value will effect program parameters. Only change this value if you understand what effect this will have.';
	sEditTitle 		: STRING := 'CAUTION';
	sDescTitle		: STRING := 'Description';
	sConvHeightMsg 	: STRING(1024) := 'Table height from ground to top of table to recieve spa from conveyor';
	sClampHeightMsg : STRING(1024) := 'Table height from ground to top of table so that spa lip is even with clamp frame for centering'; 
	sDownHeightMsg : STRING(1024) := 'Table height from gount to top of table when the table is all the way down';
	sCenterTorqueMsg : STRING(1024) := 'Torque width motors move to when centering the spa';
	sClampOnTorqueMsg : STRING(1024) := 'Torque clamp motors use when clamping onto spa lip';
	sClampOpenDistMsg : STRING(1024) := 'Distance between clamp frame jaws when opened all the way';
	sLftRotHomeSetMsg : STRING(1024) := 'Offset counts set on the motor when homing is complete';
	sRhtRotHomeSetMsg : STRING(1024) := 'Offset counts set on the motor when homing is complete';
	
	// === ERROR LOGGING ===
	aErrorData				: ARRAY[1..5,1..23] OF STRING;
	nErrorDataRow			: INT := 1;
	//Custom Errors
	sBlock	: STRING;
	sLoc	: STRING;
	nID		: UDINT;
	sMsg 	: STRING;
	
	bFlashSaveBtn 	: BOOL;
	bSaveBtnFlashOn : BOOL;
	bSaveBtn 		: BOOL;
	
	bResetMachine: BOOL;
END_VAR

// ---- GVLs/GVL_persistent.TcGVL
VAR_GLOBAL PERSISTENT
// === MACHINE SETTINGS ===
	fClampHomingTorque 		: REAL;
	fRotationHomingTorque 	: REAL;
	fTableConveyorHeight 	: REAL := 32.75; 	//Table height to recieve from conveyor
	fTableClampHeight 		: REAL := 48.5; 	// Table height to clear bottom clamp 
	fTableHomeHeight 		: REAL := 33.5; 		// Table height to send spa to centering
	fTableDownHeight		: REAL := 15.85;	// Table height when down all the way
	fCenteringTorque 		: REAL := 20; 		// % of Torque to center spa
	fClampOnTorque 			: REAL := 27;		//% of Torque to clamp onto spa
	fClampOpenDist			: REAL := 6.5;		//Distance to which the clamp is open and clears the lip of the spa
	fLftRotationHomePos 	: REAL := -66.14;	//Counts set to motor after homing to torque complete. Set in motorsInit Program.
	fRhtRotationHomePos		: REAL := 63.1;		//Counts set to motor after homing to torque complete
	fTempLftClampTorque		: REAL := 15; // Temporary Clamping for lft clamp until flange nuts are replaced

END_VAR

// ---- POUs/PROGRAMS/MAIN.TcPOU
PROGRAM MAIN
VAR
	// === SAFETY HANDLING === //
	eSafetyState 	: E_safetyState := INIT; //Current State of Safety Program in 'safetyHandler()' method
	bSafetyInit 	: BOOL; //Initialization of safety program
	sSafetyResetMsg : STRING := ''; //Msg to display the device that triggered the safety protocol
	bDispSafetyResetMsg : BOOL; //Whether or not to disp the safety screen
	nDispSafetyMsgCount : INT;
	bSafetyResetBtn : BOOL;
	bClearSafetyScrn : BOOL;
	bSafetyFaultAck : BOOL;
	fbSafetyBypassTim 	: TON; //Timer to trigger reminder that safety is currently bypassed
	fbSafetyBypassTrig 	: R_TRIG;
	fbEstopTrig			: R_TRIG;
	bBypassResetEstop 	: BOOL;
	bHideLtCurtainDisable 	: BOOL;
	fbLftCurtTrig			: R_TRIG; // Trigger for Lft Curtain Safety Buzzer Timer
	fbLftCurtTim 			: TON; //Timer to run Lft Curtain Safety Buzzer
	
	fbPageExit 		: R_TRIG;
	fbErrorPresent	: R_TRIG;
	
	
	//Used for ignition client count in "updateIgnition"
	i : INT;
	nCount : INT;
	
	//Ignition Client Handling
	fbIgnitionClientHandler : FB_ignitionClientHandler;
	
	fbFlash : TON;
	fbWritePeristentData : FB_WritePersistentData;
	
	fbRestart : TC_Restart;
END_VAR

// === SETUP PARAMETERS ===


// === CYCLIC CALLS ===
safetyHandler();
eflex();
updateIgnition(); 
updateMotors();
fbErrorPresent(CLK := GVL_machine.bErrorPresent);
IF fbErrorPresent.Q THEN
	GVL_machine.bDispErrorIcon := TRUE;
END_IF
IF GVL_machine.bErrorPresent THEN
	errorHandling();
END_IF

// === Safety Handler Output ===
bDispSafetyResetMsg := (sSafetyResetMsg <> '');
fbSafetyBypassTrig(CLK := GVL_machine.bSafetyBypass);

IF bDispSafetyResetMsg AND eSafetyState <> BYPASS THEN
	nDispSafetyMsgCount := nDispSafetyMsgCount + 1;
	IF nDispSafetyMsgCount > 50 THEN
		VisuElems.CurrentVisu := 'safetyResetScreen';
	END_IF
ELSE
	nDispSafetyMsgCount := 0;
END_IF

IF bClearSafetyScrn OR fbSafetyBypassTrig.Q THEN
	GVL_machine.bMotorsInitialized := FALSE;
	bClearSafetyScrn := FALSE;
	(*CASE GVL_machine.nPageIndex OF 
		0: VisuElems.CURRENTVISU := 'mainScreen';
		5: VisuElems.CURRENTVISU := 'manualScreen';
		10: VisuElems.CURRENTVISU := 'eflexScreen';
	END_CASE*)
	
	GVL_machine.bPageChange := TRUE;
	VisuElems.CURRENTVISU := 'mainScreen';
	GVL_machine.nPageIndex := 0;
END_IF

GVL_devices.fbTable.tempSteadyState();

IF eSafetyState = BYPASS THEN
	fbSafetyBypassTim(IN := TRUE, PT := T#5M);
	IF fbSafetyBypassTim.Q THEN 
		VisuElems.CURRENTVISU := 'safetyDisableWarning';
	END_IF
ELSE
	fbSafetyBypassTim(IN := FALSE);
END_IF

IF GVL_machine.bMuteSafety AND NOT GVL_machine.bSafetyBypass THEN
	bHideLtCurtainDisable := TRUE;
ELSE
	bHideLtCurtainDisable := FALSE;
END_IF

// === Ignition Client Handler ====
fbIgnitionClientHandler(
	sRequestedID := GVL_ignition.sReqID,
	sRequestedRole := GVL_ignition.sRole,
	sRemoveID := GVL_ignition.sRemoveID);

IF fbIgnitionClientHandler.bSessionAddError THEN
	GVL_ignition.bClientAddError := TRUE;
ELSIF fbIgnitionClientHandler.bSessionAdded THEN
	GVL_ignition.sReqID := '';
	GVL_ignition.sRole := '';
END_IF

IF fbIgnitionClientHandler.bSessionRemoved THEN
	GVL_ignition.sRemoveID := '';
END_IF

// === Page Events ===
fbPageExit.CLK := GVL_machine.bPageChange;

// === Default Light Status ===
IF NOT GVL_devices.fbLtCurtains.curtainsMuted OR NOT GVL_machine.bSafetyOk THEN
	GVL_devices.fbLtBars.redOn();
ELSE
	GVL_devices.fbLtBars.greenOn();
END_IF

IF GVL_machine.bMuteSafety THEN
	GVL_devices.fbLtCurtains.mute();
	GVL_devices.fbLtBars.yellowOn();
ELSE
	GVL_devices.fbLtCurtains.unmute();
END_IF

IF GVL_machine.bSafetyBypass THEN
	GVL_devices.fbLtBars.yellowOn();
END_IF
// === CHECK MOTOR INIT AND SAFETY ===
IF eSafetyState = OK OR eSafetyState = BYPASS THEN
	IF GVL_machine.bMotorsInitialized THEN
		//Program Steady State
		GVL_devices.fbLftWidthMotor.motorIdle := TRUE;
		GVL_devices.fbRhtWidthMotor.motorIdle := TRUE;
		GVL_devices.fbLftClampMotor.motorIdle := TRUE;
		GVL_devices.fbRhtClampMotor.motorIdle := TRUE;
		GVL_devices.fbLftRotationMotor.motorIdle := TRUE;
		GVL_devices.fbRhtRotationMotor.motorIdle := TRUE;
		GVL_devices.fbColumn0Motor.motorIdle := TRUE;
		GVL_devices.fbColumn1Motor.motorIdle := TRUE;
		GVL_devices.fbColumn2Motor.motorIdle := TRUE;
		GVL_devices.fbColumn3Motor.motorIdle := TRUE;
		
		
		
		IF fbPageExit.Q THEN
			decoupleMotors();
		END_IF
		IF GVL_machine.nPageIndex <> GVL_machine.nPrevPageIndex THEN
			GVL_machine.bPageChange := TRUE;
			GVL_machine.nPrevPageIndex := GVL_machine.nPageIndex;
		END_IF
		CASE GVL_machine.nPageIndex OF 
			5:// Run Manual Page
				manual();
			10://Run Auto Mode
				auto();
			20://Run Multi Control Mode
				multiControl();
		END_CASE
	ELSE
		//Initialize Motors
		motorsInit();
	END_IF
ELSE
	GVL_machine.bMotorsInitialized := FALSE;
END_IF

// ==== SAVE PERSISTENT VARS === //
IF GVL_machine.bFlashSaveBtn THEN
	fbFlash(IN := TRUE,PT := T#1S);
	IF fbFlash.Q THEN
		GVL_machine.bSaveBtnFlashOn := NOT GVL_machine.bSaveBtnFlashOn;
		fbFlash(IN := FALSE);
	END_IF
END_IF

IF GVL_machine.bSaveBtn THEN
	fbWritePeristentData(
	NETID:= , 
	PORT:= 851, 
	START:= TRUE, 
	TMOUT:= T#3S, 
	MODE:= SPDM_2PASS, 
	BUSY=> , 
	ERR=> , 
	ERRID=> );
	GVL_machine.bSaveBtn := FALSE;
	GVL_machine.bFlashSaveBtn := FALSE;
END_IF

// === TWINCAT RESET === //
IF GVL_machine.bResetMachine THEN
	fbRestart(
	NETID:= , 
	RESTART:= TRUE, 
	TMOUT:= T#3S, 
	BUSY=> , 
	ERR=> , 
	ERRID=> );
END_IF

METHOD decoupleMotors : BOOL
VAR_INPUT
END_VAR
GVL_devices.fbColumn0Motor.decoupleAxis();
GVL_devices.fbColumn1Motor.decoupleAxis();
GVL_devices.fbColumn2Motor.decoupleAxis();
GVL_devices.fbColumn3Motor.decoupleAxis();
GVL_devices.fbLftClampMotor.decoupleAxis();
GVL_devices.fbRhtClampMotor.decoupleAxis(); 
GVL_devices.fbLftWidthMotor.decoupleAxis();
GVL_devices.fbRhtWidthMotor.decoupleAxis();
GVL_devices.fbLftRotationMotor.decoupleAxis();
GVL_devices.fbRhtRotationMotor.decoupleAxis();
END_METHOD

METHOD safetyHandler : BOOL
VAR_INPUT
END_VAR
CASE eSafetyState OF 
	INIT:
		GVL_machine.bRunSafety := FALSE;
		IF GVL_machine.bOtherErr = FALSE THEN
			eSafetyState := PREOP;
		END_IF
		IF GVL_machine.bSafetyErrorAck THEN
			GVL_machine.bSafetyErrorAck := FALSE;
			eSafetyState := PREOP;
		END_IF
	PREOP: 
		GVL_machine.bRunSafety := TRUE;
		IF GVL_machine.bOtherErr = TRUE THEN
			GVL_machine.bSafetyErrorAck := TRUE;
			eSafetyState := INIT;
		END_IF
		IF GVL_machine.bInRun AND GVL_machine.bInRun THEN
			GVL_devices.fbLtCurtains.resetLftCurtainFB := TRUE;
			GVL_devices.fbLtCurtains.resetRhtCurtainFB := TRUE;
			GVL_devices.fbLtCurtains.enableLftCurtain := TRUE;
			GVL_devices.fbLtCurtains.enableRhtCurtain := TRUE;
			GVL_devices.fbEstop.resetEstopFB := TRUE;
			//bSafetyInit := TRUE;
			//eSafetyState := OK;
		END_IF
		IF GVL_devices.fbEstop.nEstopFbState = 6 AND GVL_devices.fbLtCurtains.nLftCurtainFbState= 6 AND GVL_devices.fbLtCurtains.nRhtCurtainFbState = 6 THEN
			GVL_devices.fbLtCurtains.resetLftCurtainFB := FALSE;
			GVL_devices.fbLtCurtains.resetRhtCurtainFB := FALSE;
			GVL_devices.fbLtCurtains.enableLftCurtain := FALSE;
			GVL_devices.fbLtCurtains.enableRhtCurtain := FALSE;
			GVL_devices.fbEstop.resetEstopFB := FALSE;
			bSafetyInit := TRUE;
			eSafetyState := OK;
		END_IF
	OK:
		//pass
	FAULT: 
		IF GVL_machine.bFbErr THEN
			sSafetyResetMsg := 'There is a Function Block Error in the Safety Program';
		ELSIF GVL_machine.bComErr THEN
			sSafetyResetMsg := 'There is a Commnunication Error in the Safety Program';
		ELSE
			sSafetyResetMsg := 'There is a Other Error in the Safety Program';
		END_IF
		IF bSafetyResetBtn THEN
			eSafetyState := RESETTING;
			bSafetyFaultAck := TRUE;
		END_IF
	WAITRESET:
		GVL_machine.bSafetyErrorAck := FALSE;
		bSafetyFaultAck := FALSE;
	RESETTING:
		GVL_machine.bSafetyErrorAck := TRUE;
		eSafetyState := WAITRESET;
	BYPASS:
		//pass
	LOCKOUT:
		//pass 
END_CASE

IF bSafetyInit THEN
	fbEstopTrig(CLK := NOT GVL_devices.fbEstop.bEstopSigOk);
	IF fbEstopTrig.Q THEN
		GVL_machine.bSafetyBypass := FALSE;
	END_IF
	IF GVL_machine.bSafetyBypass AND GVL_devices.fbEstop.bEstopSigOk THEN
		eSafetyState := BYPASS;
	ELSE
		IF GVL_machine.bFbErr OR GVL_machine.bComErr OR GVL_machine.bOtherErr THEN
			IF NOT bSafetyFaultAck THEN
				eSafetyState := FAULT;
			END_IF
		END_IF
		
		IF GVL_machine.bFbRun AND GVL_machine.bInRun THEN
			IF GVL_devices.fbEstop.nEstopFbState = 1 AND GVL_devices.fbLtCurtains.nLftCurtainFbState = 1 AND GVL_devices.fbLtCurtains.nRhtCurtainFbState = 1 THEN
				eSafetyState := OK;
				sSafetyResetMsg := '';
			END_IF	
		END_IF
		
		IF NOT GVL_machine.bSafetyOk THEN
			//A devices was triggered
			eSafetyState := ENGAGED;
			IF NOT GVL_devices.fbEstop.bEstopSigOk THEN
				sSafetyResetMsg := 'Estop: Remove Estop and Reset';
				IF bSafetyResetBtn OR bBypassResetEstop THEN
					CASE GVL_devices.fbEstop.nEstopFbState OF 
						2,3: // Triggered
							GVL_devices.fbEstop.resetEstopFB := TRUE;
						6: // Reset
							GVL_devices.fbEstop.resetEstopFB := FALSE;
							bSafetyResetBtn := FALSE;
							bBypassResetEstop := FALSE;
							sSafetyResetMsg := '';
							bClearSafetyScrn := TRUE;
					END_CASE
				END_IF
			ELSIF NOT GVL_devices.fbLtCurtains.bLftCurtainSigOk THEN
				sSafetyResetMsg := 'Left Curtain: Remove Obstruction and Reset';
				IF bSafetyResetBtn THEN
					CASE GVL_devices.fbLtCurtains.nLftCurtainFbState OF
						2,3:// Triggered
							GVL_devices.fbLtCurtains.resetLftCurtainFB := TRUE;
							GVL_devices.fbLtCurtains.enableLftCurtain := FALSE;
						6:// Reset
							GVL_devices.fbLtCurtains.resetLftCurtainFB := FALSE;
							GVL_devices.fbLtCurtains.enableLftCurtain := TRUE;
							bSafetyResetBtn := FALSE;
							sSafetyResetMsg := '';
							bClearSafetyScrn := TRUE;
					END_CASE
				END_IF
			ELSIF NOT GVL_devices.fbLtCurtains.bRhtCurtainSigOk THEN
				sSafetyResetMsg := 'Right Curtain: Remove Obstruction and Reset';
				IF bSafetyResetBtn THEN
					CASE GVL_devices.fbLtCurtains.nRhtCurtainFbState OF
						2,3:// Triggered
							GVL_devices.fbLtCurtains.resetRhtCurtainFB := TRUE;
							GVL_devices.fbLtCurtains.enableRhtCurtain := FALSE;
						6:// Reset
							GVL_devices.fbLtCurtains.resetRhtCurtainFB := FALSE;
							GVL_devices.fbLtCurtains.enableRhtCurtain := TRUE;
							bSafetyResetBtn := FALSE;
							sSafetyResetMsg := '';
							bClearSafetyScrn := TRUE;
					END_CASE
				END_IF
			END_IF
		END_IF
	END_IF
	
	// === Safety Buzzer Handling === //
	fbLftCurtTim();
	fbLftCurtTrig();
	fbLftCurtTim.PT := T#6S;
	fbLftCurtTrig.CLK := NOT GVL_devices.fbLtCurtains.bLftCurtainSigOk;
	IF fbLftCurtTrig.Q THEN
		fbLftCurtTim.IN := TRUE;
		GVL_devices.safetyBuzzer := TRUE;
	END_IF
	
	IF fbLftCurtTim.Q THEN
		fbLftCurtTim.IN := FALSE;
		GVL_devices.safetyBuzzer := FALSE;
	END_IF
END_IF
END_METHOD

METHOD updateIgnition : BOOL
VAR_INPUT
END_VAR
GVL_ignition.fClampHeight := (GVL_devices.fbLftClampMotor.distance/25.4);
GVL_ignition.fColumnHeight := -(GVL_devices.fbColumn0Motor.distance/25.4);
GVL_ignition.fTableHeight := GVL_devices.fbtable.tableHeight;
GVL_ignition.fWidthDistance := (GVL_devices.fbLftWidthMotor.distance/25.4);
GVL_ignition.fRotationDistance := GVL_devices.fbRhtRotationMotor.distance;

nCount := 0;
FOR i:=0 TO 9 DO
	IF GVL_ignition.aIgnitionClients[i].bActive THEN
		nCount := nCount + 1; 
	END_IF
END_FOR
GVL_ignition.nNumClients := nCount;
END_METHOD

END_PROGRAM

// ---- POUs/FUNCTIONS/FB_ignitionClientHandler.TcPOU
FUNCTION_BLOCK FB_ignitionClientHandler
VAR_INPUT
	sRequestedID 	: STRING(64); //New Session ID to insert
	sRequestedRole 	: STRING(32); //Role associated with new session
	sRemoveID 		: STRING(64); //Session ID to remove
END_VAR

VAR_OUTPUT
	bSessionAdded 			: BOOL;	//TRUE for 1 cycle if session added
	bSessionRemoved 		: BOOL; //TRUE for 1 cycle if session removed
	bSessionAddError 		: BOOL;
	bSessionRemoveError 	: BOOL;
END_VAR

VAR
	bPrevInsertBusy : BOOL; //Edge Detection
	bPrevRemoveBusy : BOOL;  //Edge Detection 
	bAlreadyExists : BOOL;	//Insert already exist
	i: INT;
	bOwnerExists : BOOL;
END_VAR

// Reset Outputs
bSessionAdded := FALSE;
bSessionRemoved := FALSE;

// === INSERT SESSION ===
IF sRequestedID <> '' AND NOT bPrevInsertBusy THEN
	bAlreadyExists := FALSE;
	FOR i:=0 TO 9 DO
		IF GVL_ignition.aIgnitionClients[i].bActive AND GVL_ignition.aIgnitionClients[i].sSessionId = sRequestedID THEN
			bAlreadyExists := TRUE;
			EXIT;
		END_IF
	END_FOR
	
	IF NOT bAlreadyExists THEN
		FOR i:=0 TO 9 DO
			IF NOT GVL_ignition.aIgnitionClients[i].bActive THEN
				GVL_ignition.aIgnitionClients[i].sSessionID := sRequestedID;
				GVL_ignition.aIgnitionClients[i].sRole := sRequestedRole;
				GVL_ignition.aIgnitionClients[i].bActive := TRUE;
				bSessionAdded := TRUE;
				EXIT;
			END_IF
		END_FOR
		
		IF NOT bSessionAdded THEN
			bSessionAddError := TRUE;
		END_IF
	END_IF
END_IF

IF NOT GVL_ignition.bControlAssigned AND GVL_ignition.sMachineHMISessionID <> '' THEN
	FOR i := 0 TO 9 DO
		IF GVL_ignition.aIgnitionClients[i].sSessionId = GVL_ignition.sMachineHMISessionID THEN
			GVL_ignition.aIgnitionClients[i].bHasControl := TRUE;
			GVL_ignition.bControlAssigned := TRUE;
			EXIT;
		END_IF
	END_FOR
END_IF

bPrevInsertBusy := (sRequestedID <> '');

// === REMOVE SESSION ===
IF sRemoveID <> '' AND NOT bPrevRemoveBusy THEN
	FOR i:=0 TO 9 DO
		IF GVL_ignition.aIgnitionClients[i].sSessionID = sRemoveID THEN
			GVL_ignition.aIgnitionClients[i].sSessionID := '';
			GVL_ignition.aIgnitionClients[i].sRole := '';
			GVL_ignition.aIgnitionClients[i].bActive := FALSE;
			GVL_ignition.aIgnitionClients[i].bHasControl := FALSE;
			bSessionRemoved := TRUE;
			EXIT;
		END_IF
	END_FOR
	
	IF NOT bSessionRemoved THEN
		bSessionRemoveError := TRUE;
	END_IF
END_IF

bPrevRemoveBusy := (sRemoveID <> '');

// === CURRENT SESSION IN CONTROL ===
FOR i:=0 TO 9 DO
	IF GVL_ignition.aIgnitionClients[i].bHasControl THEN
		GVL_ignition.sOwnerSessionID := GVL_ignition.aIgnitionClients[i].sSessionId;
		EXIT;
	END_IF
END_FOR

// === CLIENT CONTROL REQUEST ===
IF GVL_ignition.bTransferRequested AND GVL_ignition.bTransferApproved THEN
	FOR i:=0 TO 9 DO
		IF GVL_ignition.aIgnitionClients[i].sSessionId = GVL_ignition.sOwnerSessionID THEN
			GVL_ignition.aIgnitionClients[i].bHasControl := FALSE;
			EXIT;
		END_IF
	END_FOR
	FOR i:=0 TO 9 DO
		IF GVL_ignition.aIgnitionClients[i].sSessionId = GVL_ignition.sPendingSessionID THEN
			GVL_ignition.aIgnitionClients[i].bHasControl := TRUE;
			EXIT;
		END_IF
	END_FOR
	GVL_ignition.bTransferRequested := FALSE;
	GVL_ignition.bTransferApproved := FALSE;
	GVL_ignition.sPendingSessionID := '';
	IF GVL_ignition.sRequestedMode = 'auto' THEN
		GVL_machine.nPageIndex := 10;
	ELSIF GVL_ignition.sRequestedMode = 'manual' THEN
		GVL_machine.nPageIndex := 5;
	END_IF
	GVL_ignition.bTransferComplete := TRUE;
ELSIF GVL_ignition.bTransferRequested THEN
	bOwnerExists := FALSE;
	FOR i:=0 TO 9 DO
		IF GVL_ignition.aIgnitionClients[i].bHasControl THEN
			bOwnerExists := TRUE;
			EXIT;
		END_IF
	END_FOR
	IF NOT bOwnerExists THEN
		GVL_ignition.bTransferApproved := TRUE;
	END_IF
END_IF

END_FUNCTION_BLOCK

// ---- POUs/PROGRAMS/auto.TcPOU
PROGRAM auto
VAR
	//Program
	eState 				: E_autoState;
	ePrevState 			: E_autoState;
	eResetState			: E_resetAutoState;
	nMoveRotationState 	: INT;
	nMoveColumnState 	: INT;
	nHomeMachineState	: INT;
	fbExecuteStop 		: R_TRIG;
	
	aMoveFinish			: ARRAY[0..10] OF BOOL; // Can track the completion of up to 10 simultaneous moves
	aMoveFinishSecond   : ARRAY[0..10] OF BOOL; // Can track the completion of up to 10 simultaneous moves
	fTempRhtWidthMove 	: REAL;
	fTempLftWidthMove 	: REAL;
	
	fbMoveDelayTim		: TON;
	fbMoveDelayTimRot	: TON;

	//HMI
	bConfirmBtn 		: BOOL;
	bHideConfirmBtn 	: BOOL;
	bStartBtn			: BOOL;
	bHideStartBtn 		: BOOL;
	bStopBtn			: BOOL;
	bHideStopBtn		: BOOL;
	bResetBtn			: BOOL;
	sPromptDisp 		: STRING;
	sSetPromptDisp		: STRING;
	sCheckDisp			: STRING;
	bHideCheckDisp 		: BOOL := TRUE;
	fbProcessTimer		: TON;
	bProcessTimerIn     : BOOL;
	tProcessTimerPt		: TIME := T#3M;
	
	bShowEflex 			: BOOL;
	bShowAnimation 		: BOOL := TRUE;
	bDispContinueProg 	: BOOL;
	bContinueProgBtn 	: BOOL;
	bRestartProgBtn 	: BOOL;
	nFrameDisp 			: INT;
END_VAR

///////////////////////// PAGE CHANGE TO AUTO //////////////////////////////
IF GVL_machine.bPageChange THEN 
	F_checkMoveFinish(aMoveFinish,0,TRUE);
	bShowAnimation := TRUE;
	bShowEflex := FALSE;
	
	IF eState = CONFIRMINITHOMING THEN
		GVL_eflex.sSpaModel 	:= '';
		GVL_eflex.bEflexPresent := FALSE; 
		GVL_machine.bPageChange	:= FALSE;
	ELSE
		bDispContinueProg := TRUE;
	END_IF
END_IF

///////////////////////// AUTO STEADY STATE //////////////////////////////
IF GVL_machine.bMuteSafety OR GVL_machine.bSafetyBypass THEN
	//pass - default is yellow
ELSIF GVL_devices.fbLtCurtains.curtainsMuted THEN
	GVL_devices.fbLtBars.greenOn();
ELSE
	GVL_devices.fbLtBars.redOn();
END_IF
//bHideWarningDisp  	:= TRUE; 	bHideResetBtn 	 	:= FALSE; 
bHideStopBtn		:= FALSE;	
bHideConfirmBtn 	:= TRUE;
bHideStartBtn 	 	:= TRUE; 	
nFrameDisp 			:= 0;
sPromptDisp := '';
fbExecuteStop(CLK := bStopBtn);
//GVL_machine.bBypassMoveLimits := FALSE;
//VisuElems.CurrentVisu := 'autoScreen';	

///////////////////////// AUTO PROG //////////////////////////////////////
IF NOT bDispContinueProg THEN
	CASE eState OF 
		CONFIRMINITHOMING:
			sPromptDisp := 'Safe to home?';
			nFrameDisp := 0;
			GVL_devices.fbLtCurtains.mute();
			bHideConfirmBtn 	:= FALSE;
			IF bConfirmBtn THEN
				ePrevState := eState;
				eState := INITHOMING;
			END_IF
			
		INITHOMING:
			sPromptDisp := 'Homing';
			IF homeMachine() THEN
				
				ePrevState := eState;
				eState := SCANEFLEX;
			END_IF
			
		SCANEFLEX:
			sPromptDisp := 'Scan Eflex';
			nFrameDisp := 7;
			GVL_devices.fbLtCurtains.mute();
			tempEflex();
			IF GVL_eflex.bEflexPresent THEN 
				bHideConfirmBtn := FALSE;
				sPromptDisp := 'Confirm Scan';
				IF bConfirmBtn THEN
					GVL_eflex.bEflexPresent := FALSE; 
					ePrevState := eState;
					eState := CONFIRMPROGRAM;
				END_IF
			END_IF
		
		CONFIRMPROGRAM:
			sPromptDisp := 'Check Program, Select Start';
			GVL_devices.fbLtCurtains.mute();
			bHideStartBtn := FALSE;
			IF bStartBtn THEN
				bStartBtn := FALSE;
				ePrevState := eState;
				eState := TABLETOCONVEYOR;
			END_IF
			
		TABLETOCONVEYOR:
			sPromptDisp := 'Moving Table';
			IF GVL_devices.fbTable.moveTo(GVL_persistent.fTableConveyorHeight) THEN
				ePrevState := eState;
				eState := CONFIRMLOADED;
			END_IF
			
		CONFIRMLOADED: 
			sPromptDisp := 'Confirm Spa Loaded';
			nFrameDisp := 2;
			GVL_devices.fbLtCurtains.mute();
			bHideConfirmBtn := FALSE;
			IF bConfirmBtn THEN
				ePrevState := eState;
				eState := TABLETOCLAMP;
			END_IF
		
		TABLETOCLAMP:
			sPromptDisp := 'Raising Table';
			IF GVL_devices.fbTable.moveTo(GVL_persistent.fTableClampHeight - 1) THEN
				ePrevState := eState;
				eState := CENTERSPA;
			END_IF
			
		CENTERSPA:
			sPromptDisp := 'Centering Spa';
			IF NOT aMoveFinish[0] THEN
				CASE GVL_devices.fbLftWidthMotor.moveToTorque('NULL',GVL_persistent.fCenteringTorque,0) OF 
					1:// Done
						aMoveFinish[0] := TRUE;
					13:// Error
						GVL_machine.motorErrorList := LFTWIDTH;
						GVL_machine.bErrorPresent := TRUE;
				END_CASE
			END_IF
			IF NOT aMoveFinish[1] THEN
				CASE GVL_devices.fbRhtWidthMotor.moveToTorque('NULL',-GVL_persistent.fCenteringTorque,0) OF 
					1:// Done
						aMoveFinish[1] := TRUE;
					13:// Error
						GVL_machine.motorErrorList := RHTWIDTH;
						GVL_machine.bErrorPresent := TRUE;
				END_CASE
			END_IF
			
			IF F_checkMoveFinish(aMoveFinish,2,FALSE) THEN
				F_checkMoveFinish(aMoveFinish,0,TRUE);
				ePrevState := eState;
				eState := OPENCLAMP;
			END_IF
			
		OPENCLAMP: 
			sPromptDisp := 'Opening Clamps';
			IF NOT aMoveFinish[0] THEN
				fTempRhtWidthMove := (ABS(GVL_devices.fbRhtWidthMotor.fbMotor.NcToPlc.ActPos)/25.4)- 2;
				aMoveFinish[0] := TRUE;
			END_IF
			IF NOT aMoveFinish[1] THEN
				fTempLftWidthMove := (ABS(GVL_devices.fbLftWidthMotor.fbMotor.NcToPlc.ActPos)/25.4)- 2;
				aMoveFinish[1] := TRUE;
			END_IF
			IF NOT aMoveFinish[2] THEN
				CASE GVL_devices.fbLftWidthMotor.moveTo('NULL',fTempLftWidthMove) OF 
					1:// Done
						IF fTempLftWidthMove < GVL_devices.fbLftWidthMotor.distance + 0.5 OR fTempLftWidthMove > GVL_devices.fbLftWidthMotor.distance - 0.5 THEN
							aMoveFinish[2] := TRUE;
						END_IF
					13: //Error
						GVL_machine.motorErrorList := LFTWIDTH;
						GVL_machine.bErrorPresent := TRUE;
					15: //Halfway 
						aMoveFinish[6] := TRUE;
				END_CASE
			END_IF
			IF NOT aMoveFinish[3] THEN
				CASE GVL_devices.fbRhtWidthMotor.moveTo('NULL',fTempRhtWidthMove) OF 
					1:// Done
						aMoveFinish[3] := TRUE;
					13:// Error
						GVL_machine.motorErrorList := RHTWIDTH;
						GVL_machine.bErrorPresent := TRUE;
					15: //Halfway 
						aMoveFinish[7] := TRUE;
				END_CASE
			END_IF
			IF aMoveFinish[6] AND NOT aMoveFinish[4] THEN
				(*CASE GVL_devices.fbLftClampMotor.moveTo('NULL',GVL_persistent.fClampOpenDist) OF 
					1:// Done
						aMoveFinish[4] := TRUE;
					13://Error
						GVL_machine.motorErrorList := LFTCLAMP;
						GVL_machine.bErrorPresent := TRUE;
				END_CASE*)
				IF GVL_devices.fbLftClampMotor.tempCylinderOpen() THEN
					aMoveFinish[4] := TRUE;
				END_IF
			END_IF
			IF aMoveFinish[7] AND NOT aMoveFinish[5] THEN
				CASE GVL_devices.fbRhtClampMotor.moveTo('NULL',GVL_persistent.fClampOpenDist) OF 
					1:// Done
						aMoveFinish[5] := TRUE;
					13://Error
						GVL_machine.motorErrorList := RHTCLAMP;
						GVL_machine.bErrorPresent := TRUE;
				END_CASE
			END_IF
			IF F_checkMoveFinish(aMoveFinish,8,FALSE) THEN
				F_checkMoveFinish(aMoveFinish,0,TRUE);
				ePrevState := eState;
				eState := MOVETOCLAMP;
			END_IF
			
		MOVETOCLAMP:
			sPromptDisp := 'Moving Clamps In';

			IF NOT aMoveFinish[3] THEN 
				IF GVL_devices.fbTable.moveTo(GVL_persistent.fTableClampHeight) THEN
					aMoveFinish[3] := TRUE;
				END_IF
			END_IF
			IF aMoveFinish[3] THEN
				IF NOT aMoveFinish[0] THEN
					CASE GVL_devices.fbLftWidthMotor.moveToSensor(1) OF 
						1:// Done
							aMoveFinish[0] := TRUE;
						13:// Error
							GVL_machine.motorErrorList := LFTWIDTH;
							GVL_machine.bErrorPresent := TRUE;
					END_CASE
				END_IF
				IF NOT aMoveFinish[1] THEN
					CASE GVL_devices.fbRhtWidthMotor.moveToSensor(1) OF 
						1:// Done
							aMoveFinish[1] := TRUE;
						13://Error
							GVL_machine.motorErrorList := RHTWIDTH;
							GVL_machine.bErrorPresent := TRUE;
					END_CASE
				END_IF
			END_IF
			IF aMoveFinish[0] AND aMoveFinish[1] THEN
				IF NOT aMoveFinish[2] THEN
					IF GVL_devices.fbTable.moveTo(GVL_persistent.fTableClampHeight - 3.5) THEN
						aMoveFinish[2] := TRUE;
					END_IF
				END_IF
			END_IF
			
 			IF F_checkMoveFinish(aMoveFinish,4,FALSE) THEN
				ePrevState := eState;
				eState := CLAMPSPA;
			END_IF
			
		CLAMPSPA:
			sPromptDisp := 'Clamping Spa';
			IF NOT aMoveFinish[0] THEN
				(*CASE GVL_devices.fbLftClampMotor.moveToTorque('NULL',GVL_persistent.fTempLftClampTorque,0) OF 
					1:// Done
						aMoveFinish[0] := TRUE;
					13:// Error
						GVL_machine.motorErrorList := LFTCLAMP;
						GVL_machine.bErrorPresent := TRUE;
				END_CASE*)
				IF GVL_devices.fbLftClampMotor.tempCylinderClose() THEN
					aMoveFinish[0] := TRUE;
				END_IF
			END_IF
			IF NOT aMoveFinish[1] THEN
				CASE GVL_devices.fbRhtClampMotor.moveToTorque('NULL',GVL_persistent.fClampOnTorque,1) OF
					1:// Done
						aMoveFinish[1] := TRUE;
					13:// Error
						GVL_machine.motorErrorList := RHTCLAMP;
						GVL_machine.bErrorPresent := TRUE;
				END_CASE
			END_IF
			(*IF NOT aMoveFinish[2] THEN
				IF GVL_devices.fbTable.moveTo(GVL_persistent.fTableClampHeight - 2) THEN
					aMoveFinish[2] := TRUE;
				END_IF
			END_IF*)
			
			IF F_checkMoveFinish(aMoveFinish,2,FALSE) THEN
				ePrevState := eState;
				//eState := ROTATESPA;
				eState := CONFIRMMANUALCLAMPING;
			END_IF
		
		CONFIRMMANUALCLAMPING:
			sPromptDisp := 'Confirm Clamp on Spa';
			nFrameDisp := 2;
			GVL_devices.fbLtCurtains.mute();
			bHideConfirmBtn := FALSE;
			IF bConfirmBtn THEN
				ePrevState := eState;
				eState := ROTATESPA;
			END_IF
			
		ROTATESPA:
			(*IF GVL_devices.fbLftClampMotor.distance > -20 THEN
				sSetPromptDisp := 'Lft clamp: $n Spa not clamped';
				ePrevState := eState;
				eState := PROGERRORSTOP;
			ELSIF GVL_devices.fbRhtClampMotor.distance < 20 THEN
				sSetPromptDisp := 'Rht clamp: $n Spa not clamped';
				ePrevState := eState;
				eState := PROGERRORSTOP;
			END_IF*)
			IF GVL_devices.fbRhtClampMotor.distance < 20 THEN
				sSetPromptDisp := 'Rht clamp: $n Spa not clamped';
				ePrevState := eState;
				eState := PROGERRORSTOP;
			END_IF
			
			sPromptDisp := 'Rotating Spa';
			IF NOT aMoveFinish[0] THEN
				CASE moveColumns('NULL',GVL_eflex.fFlipHeight,1) OF 
					1:// Done
						aMoveFinish[0] := TRUE;
						aMoveFinish[1] := TRUE;
					13:// Error
						GVL_devices.fbColumn0Motor.stop();
						GVL_devices.fbColumn1Motor.stop();
						GVL_devices.fbColumn2Motor.stop();
						GVL_devices.fbColumn3Motor.stop();
						ePrevState := ROTATESPA;
						eState := PROGERRORSTOP;
						sSetPromptDisp := 'Column Faulted Retry Start';
					15:// Move is halway
						IF GVL_devices.fbColumn0Motor.distance < -25 THEN
							aMoveFinish[1] := TRUE;
						END_IF
				END_CASE
			END_IF
			IF aMoveFinish[1] THEN
				IF NOT aMoveFinish[2] THEN
					IF GVL_devices.fbColumn0Motor.distance < -25 THEN
						CASE moveRotation('NULL',270) OF 
							1:// Done
								aMoveFinish[2] := TRUE;
							13:// Error
								GVL_devices.fbLftRotationMotor.stop();
								GVL_devices.fbRhtRotationMotor.stop();
							15:// Move Halfway	
								aMoveFinish[3] := TRUE;
						END_CASE
					END_IF
				END_IF
			END_IF
			
			IF NOT aMoveFinish[4] THEN
				IF GVL_devices.fbTable.moveTo(GVL_persistent.fTableDownHeight) THEN
					aMoveFinish[4] := TRUE;
				END_IF
			END_IF
		
			
			IF F_checkMoveFinish(aMoveFinish,5,FALSE) THEN
				ePrevState := eState;
				eState := TABLETOBASE;
			END_IF
		
		TABLETOBASE:
			sPromptDisp := 'Raising Table';
			IF GVL_devices.fbTable.moveTo(GVL_eflex.fBaseInHeight) THEN
				ePrevState := eState;
				eState := CONFIRMSKIIS;
			END_IF
			
		CONFIRMSKIIS:
			sPromptDisp := 'Remove Skiis'; 
			GVL_devices.fbLtCurtains.mute();
			bHideConfirmBtn 	:= FALSE;
			IF bConfirmBtn THEN
				bConfirmBtn := FALSE;
				ePrevState := eState;
				eState := CONFIRMBASE;
			END_IF
			
		CONFIRMBASE:
			sPromptDisp := 'Load Base';
			GVL_devices.fbLtCurtains.mute();
			bHideConfirmBtn 	:= FALSE;
			IF bConfirmBtn THEN
				bConfirmBtn := FALSE;
				ePrevState := eState;
				eState := LOWERSPA;
			END_IF
			
		LOWERSPA:
			sPromptDisp := 'Lowering Spa';
			IF NOT aMoveFinish[0] THEN 
				CASE moveColumns('NULL',GVL_eflex.fStudHeight,1) OF 
					1:// Done
						aMoveFinish[0] := TRUE;
					13:// Error
						GVL_devices.fbColumn0Motor.stop();
						GVL_devices.fbColumn1Motor.stop();
						GVL_devices.fbColumn2Motor.stop();
						GVL_devices.fbColumn3Motor.stop();
						ePrevState := LOWERSPA;
						eState := PROGERRORSTOP;
						sPromptDisp := 'Column Faulted Retry Start';
					15:// Move Halfway
						aMoveFinish[1] := TRUE;
				END_CASE
			END_IF
			
			IF NOT aMoveFinish[4] THEN
				IF GVL_devices.fbTable.moveTo(GVL_eflex.fSpaOutHeight) THEN
					aMoveFinish[4] := TRUE;
				END_IF
			END_IF
			
			IF aMoveFinish[1] THEN
				IF NOT aMoveFinish[2] THEN
					(*CASE GVL_devices.fbLftClampMotor.moveTo('NULL',9.5) OF 
						1: // Done
							aMoveFinish[2] := TRUE;
						13: // Error
							GVL_machine.motorErrorList := LFTCLAMP;
							GVL_machine.bErrorPresent := TRUE;
					END_CASE*)
					IF GVL_devices.fbLftClampMotor.tempCylinderOpen() THEN
						aMoveFinish[2] := TRUE;
					END_IF
				END_IF
				IF NOT aMoveFinish[3] THEN
					CASE GVL_devices.fbRhtClampMotor.moveTo('NULL',9.5) OF 
						1:// Done
							aMoveFinish[3] := TRUE;
						13:// Error
							GVL_machine.motorErrorList := RHTCLAMP;
							GVL_machine.bErrorPresent := TRUE;
					END_CASE
				END_IF
			END_IF
			IF F_checkMoveFinish(aMoveFinish,5,FALSE) THEN
				ePrevState := eState;
				eState := CLAMPRETURN;
			END_IF
			
		CLAMPRETURN:
			sPromptDisp := 'Clamps Moving Out';
			IF NOT aMoveFinish[0] THEN
				CASE GVL_devices.fbLftWidthMotor.homeToSensorCustom() OF
					1:// Done
						aMoveFinish[0] := TRUE;
					13:// Error
						GVL_machine.motorErrorList := LFTWIDTH;
						GVL_machine.bErrorPresent := TRUE;
				END_CASE 
			END_IF
			IF NOT aMoveFinish[1] THEN
				CASE GVL_devices.fbRhtWidthMotor.homeToSensorCustom() OF 
					1: //Done
						aMoveFinish[1] := TRUE;
					13: //Error\
						GVL_machine.motorErrorList := RHTWIDTH;
						GVL_machine.bErrorPresent := TRUE;
				END_CASE
			END_IF
			
			IF F_checkMoveFinish(aMoveFinish,2,FALSE) THEN
				ePrevState := eState;
				eState := CONFIRMSPAUNLOAD;
			END_IF
			
		CONFIRMSPAUNLOAD:
			bConfirmBtn := TRUE; // Bypass ConfirmSpaUnload Prompt
			GVL_devices.fbLtCurtains.mute();
			bHideConfirmBtn 	:= FALSE;
			sPromptDisp := 'Unload Spa';
			IF bConfirmBtn OR NOT GVL_devices.fbTable.spaLoaded THEN
				bConfirmBtn := FALSE;
				GVL_eflex.bEflexPresent := FALSE;
				GVL_eflex.fFlipHeight := 0;
				GVL_eflex.fStudHeight := 0;
				GVL_eflex.sSpaModel := '';
				ePrevState := eState;
				eState := INITHOMING;
			END_IF
			
		STOPPROGRAM:
			GVL_devices.fbLtCurtains.mute();
			sPromptDisp := 'Program Stopped';
			bHideStartBtn := FALSE;
			bHideStopBtn := TRUE;
			IF bStartBtn THEN
				sPromptDisp := 'Program Starting';
				bHideStartBtn := TRUE;
				bHideStopBtn := TRUE;
				motorsInit();
				IF motorsInit.bMotorsInit THEN
					bStartBtn := FALSE;
					bStopBtn := FALSE;
					bHideStopBtn := FALSE;
					eState := ePrevState;
				END_IF
			END_IF
			
		RESETPROGRAM:
			resetAutoProgram();
			IF eResetState = RESETDONE THEN
				sPromptDisp := 'Reset Program';
				GVL_eflex.sSpaModel 	:= '';
				GVL_eflex.bEflexPresent := FALSE;
				bDispContinueProg := FALSE;
				GVL_machine.bPageChange	:= FALSE;
				bRestartProgBtn := FALSE;
				F_checkMoveFinish(aMoveFinish,2,TRUE);
				bStartBtn := FALSE;
				bStopBtn := FALSE;
				bConfirmBtn := FALSE;
				bResetBtn := FALSE;
				eState := CONFIRMINITHOMING;
			END_IF
			
		RESETMOTORS:
			bHideConfirmBtn := TRUE;
			bHideStopBtn := TRUE;
			bHideStartBtn := TRUE;
			sPromptDisp := 'Initializing Motors';
			motorsInit();
			IF motorsInit.bMotorsInit THEN
				eState := RESETPROGRAM;
			END_IF
			
		MOTORFAULTED: 
			bHideConfirmBtn := TRUE;
			bHideStopBtn := TRUE;
			bHideStartBtn := TRUE;
			sPromptDisp := 'Motor Fault: Resetting';
			motorsInit();
			IF motorsInit.bMotorsInit THEN
				eState := ePrevState;
			END_IF
			
		PROGERRORSTOP: 
			GVL_devices.fbLtCurtains.mute();
			bHideStartBtn := FALSE;
			bHideStopBtn := TRUE;
			sPromptDisp := sSetPromptDisp;
			IF bStartBtn THEN
				sPromptDisp := 'Program Starting';
				bHideStartBtn := TRUE;
				bHideStopBtn := TRUE;
				motorsInit();
				IF motorsInit.bMotorsInit THEN
					bStartBtn := FALSE;
					bStopBtn := FALSE;
					bHideStopBtn := FALSE;
					eState := ePrevState;
				END_IF
			END_IF
			
		RESETLFTCOLUMNS:
			GVL_devices.fbLtCurtains.mute();
			bHideStartBtn := FALSE;
			bHideStopBtn := TRUE;
			sPromptDisp := sSetPromptDisp;
			IF bStartBtn THEN
				sPromptDisp := 'Program Starting';
				bHideStartBtn := TRUE;
				bHideStopBtn := TRUE;
				motorsInit();
				IF motorsInit.bMotorsInit THEN
					bStartBtn := FALSE;
					bStopBtn := FALSE;
					bHideStopBtn := FALSE;
					eState := MATCHLFTCOLUMNS;
				END_IF
			END_IF
		
		MATCHLFTCOLUMNS:
			sPromptDisp := sSetPromptDisp;
			IF ABS(GVL_devices.fbColumn0Motor.distance) < ABS(GVL_devices.fbColumn1Motor.distance) THEN
				CASE GVL_devices.fbColumn0Motor.moveTo('NULL',GVL_devices.fbColumn1Motor.distance / 25.4) OF 
					1: //Done
						eState := ePrevState;
					13: //Error
						GVL_devices.fbColumn0Motor.stop();
						GVL_devices.fbColumn1Motor.stop();
						GVL_devices.fbColumn2Motor.stop();
						GVL_devices.fbColumn3Motor.stop();
						ePrevState := INITHOMING;
						eState := PROGERRORSTOP;
						sSetPromptDisp := 'Column Faulted Retry Start';
				END_CASE
			ELSE
				CASE GVL_devices.fbColumn1Motor.moveTo('NULL',GVL_devices.fbColumn0Motor.distance / 25.4) OF 
					1: //Done
						eState := ePrevState;
					13: //Error
						GVL_devices.fbColumn0Motor.stop();
						GVL_devices.fbColumn1Motor.stop();
						GVL_devices.fbColumn2Motor.stop();
						GVL_devices.fbColumn3Motor.stop();
						ePrevState := INITHOMING;
						eState := PROGERRORSTOP;
						sSetPromptDisp := 'Column Faulted Retry Start';
				END_CASE
			END_IF
					
		RESETRHTCOLUMNS:
			GVL_devices.fbLtCurtains.mute();
			bHideStartBtn := FALSE;
			bHideStopBtn := TRUE;
			sPromptDisp := sSetPromptDisp;
			IF bStartBtn THEN
				sPromptDisp := 'Program Starting';
				bHideStartBtn := TRUE;
				bHideStopBtn := TRUE;
				motorsInit();
				IF motorsInit.bMotorsInit THEN
					bStartBtn := FALSE;
					bStopBtn := FALSE;
					bHideStopBtn := FALSE;
					eState := MATCHRHTCOLUMNS;
				END_IF
			END_IF
		
		MATCHRHTCOLUMNS:
			sPromptDisp := sSetPromptDisp;
			IF ABS(GVL_devices.fbColumn2Motor.distance) < ABS(GVL_devices.fbColumn3Motor.distance) THEN
				CASE GVL_devices.fbColumn2Motor.moveTo('NULL',GVL_devices.fbColumn3Motor.distance / 25.4) OF 
					1: //Done
						eState := ePrevState;
					13: //Error
						GVL_devices.fbColumn0Motor.stop();
						GVL_devices.fbColumn1Motor.stop();
						GVL_devices.fbColumn2Motor.stop();
						GVL_devices.fbColumn3Motor.stop();
						ePrevState := INITHOMING;
						eState := PROGERRORSTOP;
						sSetPromptDisp := 'Column Faulted Retry Start';
				END_CASE
			ELSE
				CASE GVL_devices.fbColumn3Motor.moveTo('NULL',GVL_devices.fbColumn2Motor.distance / 25.4) OF 
					1: //Done
						eState := ePrevState;
					13: //Error
						GVL_devices.fbColumn0Motor.stop();
						GVL_devices.fbColumn1Motor.stop();
						GVL_devices.fbColumn2Motor.stop();
						GVL_devices.fbColumn3Motor.stop();
						ePrevState := INITHOMING;
						eState := PROGERRORSTOP;
						sSetPromptDisp := 'Column Faulted Retry Start';
				END_CASE
			END_IF
	END_CASE
ELSE // Waiting for confirmation from operator to load previous running program or restart. 
	nFrameDisp := 8;
	IF bContinueProgBtn THEN
		bDispContinueProg := FALSE;
		GVL_machine.bPageChange	:= FALSE;
		bContinueProgBtn := FALSE;
		F_checkMoveFinish(aMoveFinish,0,TRUE);
	ELSIF bRestartProgBtn THEN
		eState := CONFIRMINITHOMING;
		GVL_eflex.sSpaModel 	:= '';
		GVL_eflex.bEflexPresent := FALSE;
		bDispContinueProg := FALSE;
		GVL_machine.bPageChange	:= FALSE;
		bRestartProgBtn := FALSE;
		F_checkMoveFinish(aMoveFinish,0,TRUE);
	END_IF
END_IF

IF bResetBtn THEN
	eResetState := CHECKWIDTH;
	eState := RESETMOTORS;
	bResetBtn := FALSE;
ELSIF bStopBtn THEN
	ePrevState := eState;
	bStopBtn := FALSE;
	eState := STOPPROGRAM;
ELSIF eState <> RESETMOTORS AND eState <> RESETPROGRAM AND eState <> STOPPROGRAM AND eState <> MOTORFAULTED AND motorFault() THEN
	ePrevState := eState;
	eState := MOTORFAULTED;
END_IF

backgroundCheck();

METHOD backgroundCheck : BOOL
VAR_INPUT
END_VAR
bHideCheckDisp := TRUE;
sCheckDisp := '';
fbProcessTimer(IN := bProcessTimerIn, PT := tProcessTimerPt);
bProcessTimerIn := FALSE;
//IF eState <> CONFIRMINITHOMING OR eState <> INITHOMING THEN
// ==== Check to see if any column motor is moving when others are not ==== //
IF eState <> RESETLFTCOLUMNS AND eState <> RESETRHTCOLUMNS AND eState <> MATCHLFTCOLUMNS AND eState <> MATCHRHTCOLUMNS AND eState <> PROGERRORSTOP THEN
	IF GVL_devices.fbColumn0Motor.distance > -1000 AND GVL_devices.fbColumn0Motor.distance < 1000 THEN
		IF ABS(GVL_devices.fbColumn0Motor.distance - GVL_devices.fbColumn1Motor.distance) > 5 THEN
			GVL_devices.fbColumn0Motor.estop();
			GVL_devices.fbColumn1Motor.estop();
			GVL_devices.fbColumn2Motor.estop();
			GVL_devices.fbColumn3Motor.estop();
			
			GVL_machine.sBlock := DINT_TO_STRING(eState);
			GVL_machine.sLoc := 'LFT Column Match';
			GVL_machine.nID := 0;
			GVL_machine.motorErrorList := CUSTOM;
			GVL_machine.bErrorPresent := TRUE;
			
			IF ABS(GVL_devices.fbColumn0Motor.distance - GVL_devices.fbColumn1Motor.distance) < 12 THEN
				ePrevState := eState;
				eState := RESETLFTCOLUMNS;
				sSetPromptDisp := 'Lft Columns: $n Counts not matching $n Start to reset.';
			ELSE
				ePrevState := eState;
				eState := PROGERRORSTOP;
				sSetPromptDisp := 'Lft Columns: $n Counts not matching. $n Maintenance required';
			END_IF
		END_IF
	END_IF
	
	IF GVL_devices.fbColumn2Motor.distance > -1000 AND GVL_devices.fbColumn2Motor.distance < 1000 THEN 
		IF ABS(GVL_devices.fbColumn2Motor.distance - GVL_devices.fbColumn3Motor.distance) > 5 THEN
			GVL_devices.fbColumn0Motor.estop();
			GVL_devices.fbColumn1Motor.estop();
			GVL_devices.fbColumn2Motor.estop();
			GVL_devices.fbColumn3Motor.estop();
			
			GVL_machine.sBlock := DINT_TO_STRING(eState);
			GVL_machine.sLoc := 'RHT Column Match';
			GVL_machine.nID := 1;
			GVL_machine.motorErrorList := CUSTOM;
			GVL_machine.bErrorPresent := TRUE;
			
			IF ABS(GVL_devices.fbColumn2Motor.distance - GVL_devices.fbColumn3Motor.distance) < 12 THEN
				ePrevState := eState;
				eState := RESETRHTCOLUMNS;
				sSetPromptDisp := 'Rht Columns: $n Counts not matching $n Start to reset.';
			ELSE
				ePrevState := eState;
				eState := PROGERRORSTOP;
				sSetPromptDisp := 'Rht Columns: $n Counts not matching $n Maintenance required';
			END_IF
		END_IF
	END_IF

	IF GVL_devices.fbColumn0Motor.fbMotor.Status.Moving OR GVL_devices.fbColumn1Motor.fbMotor.Status.Moving OR GVL_devices.fbColumn2Motor.fbMotor.Status.Moving OR GVL_devices.fbColumn3Motor.fbMotor.Status.Moving THEN
		IF GVL_devices.fbColumn0Motor.fbMotor.Status.NotMoving OR GVL_devices.fbColumn1Motor.fbMotor.Status.NotMoving OR GVL_devices.fbColumn2Motor.fbMotor.Status.NotMoving OR GVL_devices.fbColumn3Motor.fbMotor.Status.NotMoving THEN
			fbMoveDelayTim(IN := FALSE, PT := T#500MS);
			IF fbMoveDelayTim.Q THEN
				GVL_devices.fbColumn0Motor.estop();
				GVL_devices.fbColumn1Motor.estop();
				GVL_devices.fbColumn2Motor.estop();
				GVL_devices.fbColumn3Motor.estop();
				ePrevState := eState;
				eState := PROGERRORSTOP;
				sSetPromptDisp := 'Column Faulted Retry Start';
			END_IF
		END_IF
	ELSE
		fbMoveDelayTim(IN := FALSE);
	END_IF
END_IF


// === Check Software Limit Switches on Motors === //
(*IF GVL_devices.fbRhtRotationMotor.fbMotor.Status.SoftLimitMaxExceeded OR GVL_devices.fbRhtRotationMotor.fbMotor.Status.SoftLimitMinExceeded THEN
	bHideCheckDisp := FALSE;
	sCheckDisp := 'Rht rotation motor: $n Out of Range';
END_IF
IF GVL_devices.fbLftRotationMotor.fbMotor.Status.SoftLimitMaxExceeded OR GVL_devices.fbLftRotationMotor.fbMotor.Status.SoftLimitMinExceeded THEN
	bHideCheckDisp := FALSE;
	sCheckDisp := 'Lft rotation motor: $n Out of Range';
END_IF
	
IF GVL_devices.fbColumn0Motor.fbMotor.Status.SoftLimitMaxExceeded OR GVL_devices.fbColumn0Motor.fbMotor.Status.SoftLimitMinExceeded THEN
	bHideCheckDisp := FALSE;
	sCheckDisp := 'Column 0 Motor: $n Out of Range';
END_IF
IF GVL_devices.fbColumn1Motor.fbMotor.Status.SoftLimitMaxExceeded OR GVL_devices.fbColumn0Motor.fbMotor.Status.SoftLimitMinExceeded THEN
	bHideCheckDisp := FALSE;
	sCheckDisp := 'Column 1 Motor: $n Out of Range';
END_IF
IF GVL_devices.fbColumn2Motor.fbMotor.Status.SoftLimitMaxExceeded OR GVL_devices.fbColumn0Motor.fbMotor.Status.SoftLimitMinExceeded THEN
	bHideCheckDisp := FALSE;
	sCheckDisp := 'Column 2 Motor: $n Out of Range';
END_IF
IF GVL_devices.fbColumn3Motor.fbMotor.Status.SoftLimitMaxExceeded OR GVL_devices.fbColumn0Motor.fbMotor.Status.SoftLimitMinExceeded THEN
	bHideCheckDisp := FALSE;
	sCheckDisp := 'Column 3 Motor: $n Out of Range';
END_IF

IF GVL_devices.fbLftWidthMotor.fbMotor.Status.SoftLimitMaxExceeded OR GVL_devices.fbLftWidthMotor.fbMotor.Status.SoftLimitMinExceeded THEN
	bHideCheckDisp := FALSE;
	sCheckDisp := 'Lft width motor: $n Out of Range';
END_IF
IF GVL_devices.fbRhtWidthMotor.fbMotor.Status.SoftLimitMaxExceeded OR GVL_devices.fbRhtWidthMotor.fbMotor.Status.SoftLimitMinExceeded THEN
	bHideCheckDisp := FALSE;
	sCheckDisp := 'Rht width: $n Out of Range';
END_IF

IF GVL_devices.fbLftClampMotor.fbMotor.Status.SoftLimitMaxExceeded OR GVL_devices.fbLftClampMotor.fbMotor.Status.SoftLimitMinExceeded THEN
	bHideCheckDisp := FALSE;
	sCheckDisp := 'Lft clamp motor: $n Out of Range';
END_IF
IF GVL_devices.fbRhtClampMotor.fbMotor.Status.SoftLimitMaxExceeded OR GVL_devices.fbRhtClampMotor.fbMotor.Status.SoftLimitMinExceeded THEN
	bHideCheckDisp := FALSE;
	sCheckDisp := 'Rht clamp motor: $n Out of Range';
END_IF
*)
// === Check if all 4 power supplies are on === //
IF GVL_devices.fbColumn0Motor.fbMotor.Status.DriveDeviceError
OR GVL_devices.fbLftClampMotor.fbMotor.Status.DriveDeviceError
OR GVL_devices.fbColumn2Motor.fbMotor.Status.DriveDeviceError 
OR GVL_devices.fbRhtClampMotor.fbMotor.Status.DriveDeviceError THEN
	bHideCheckDisp := FALSE;
	sCheckDisp := 'No Power $n Check Motor Power Supplies';
END_IF

// ==== Check for debris under table sensor === //
IF GVL_devices.fbTable.tableHeight < GVL_persistent.fTableDownHeight - 0.10 THEN 
	bHideCheckDisp := FALSE;
	sCheckDisp := 'Table Sensor Height: $n Check debris under table';
END_IF
IF GVL_devices.fbTable.tableHeight > GVL_persistent.fTableDownHeight + 35 THEN 
	bHideCheckDisp := FALSE;
	sCheckDisp := 'Table Sensor Height: $n Check debris under table';
END_IF

// === Compare clamp distances === //
(*IF ABS(GVL_devices.fbRhtClampMotor.distance + GVL_devices.fbLftClampMotor.distance) > 20 THEN
	bHideCheckDisp := FALSE;
	sCheckDisp := 'Clamping: Clamps not aligned $n Check clamps';
END_IF*)

CASE eState OF 
	CONFIRMINITHOMING://
	INITHOMING://
	SCANEFLEX://
	CONFIRMPROGRAM://
	TABLETOCONVEYOR://
	CONFIRMLOADED://
	TABLETOCLAMP://
	CENTERSPA://
		bProcessTimerIn := TRUE;
		tProcessTimerPt := T#2S;
		IF NOT fbProcesstimer.Q AND (aMoveFinish[1] OR aMoveFinish[2]) THEN
			bHideCheckDisp := FALSE;
			sCheckDisp := 'Width Motors: $n Early torque out';
		END_IF
		IF NOT bHideCheckDisp THEN
			bHideCheckDisp := FALSE;
			sCheckDisp := 'Width Motors: $n Early torque out';
		END_IF
		
	OPENCLAMP://
		IF GVL_devices.fbLftWidthMotor.distance < 10 THEN
			bHideCheckDisp := FALSE;
			sCheckDisp := 'Lft Width Motor: $n Centering Failed';
		END_IF
		IF GVL_devices.fbRhtWidthMotor.distance < 10 THEN
			bHideCheckDisp := FALSE;
			sCheckDisp := 'Rht Width Motor: $n Centering Failed';
		END_IF
		
	MOVETOCLAMP://
		bProcessTimerIn := TRUE;
		tProcessTimerPt := T#90S;
		IF fbProcesstimer.Q THEN
			IF NOT GVL_devices.fbLftWidthMotor.bClampSensor THEN
				bHideCheckDisp := FALSE;
				sCheckDisp := 'Lft width sensor: $n Sensor timed out';
			END_IF
			IF NOT GVL_devices.fbRhtWidthMotor.bClampSensor THEN
				bHideCheckDisp := FALSE;
				sCheckDisp := 'Rht width sensor: $n Sensor timed out';
			END_IF
		END_IF
		
		IF ABS(GVL_devices.fbLftWidthMotor.fbMotor.NcToPlc.ActTorque) > ABS(GVL_devices.fbLftWidthMotor.jogTorque) THEN
			bHideCheckDisp := FALSE;
			sCheckDisp := 'Lft Width Motor: $n Torque Exceeded';
		END_IF
		IF ABS(GVL_devices.fbRhtWidthMotor.fbMotor.NcToPlc.ActTorque) > ABS(GVL_devices.fbRhtWidthMotor.jogTorque) THEN
			bHideCheckDisp := FALSE;
			sCheckDisp := 'Rht Width Motor: $n Torque Exceeded';
		END_IF
		
	CLAMPSPA://
		IF NOT GVL_devices.fbLftWidthMotor.bClampSensor THEN
			bHideCheckDisp := FALSE;
			sCheckDisp := 'Lft width sensor: $n Check spa is clamped';
		END_IF
		IF NOT GVL_devices.fbRhtWidthMotor.bClampSensor THEN
			bHideCheckDisp := FALSE;
			sCheckDisp := 'Rht width sensor: $n Check spa is clamped';
		END_IF
		
		(*IF GVL_devices.fbLftClampMotor.distance > -20 THEN
			bHideCheckDisp := FALSE;
			sCheckDisp := 'Lft clamp: $n Spa not clamped';
		END_IF*)
		IF GVL_devices.fbRhtClampMotor.distance < 20 THEN
			bHideCheckDisp := FALSE;
			sCheckDisp := 'Rht clamp: $n Spa not clamped';
		END_IF
		
		
	ROTATESPA://
		(*IF GVL_devices.fbLftClampMotor.distance > -20 THEN
			bHideCheckDisp := FALSE;
			sCheckDisp := 'Lft clamp: $n Spa not clamped';
		END_IF*)
		IF GVL_devices.fbRhtClampMotor.distance < 20 THEN
			bHideCheckDisp := FALSE;
			sCheckDisp := 'Rht clamp: $n Spa not clamped';
		END_IF
	TABLETOBASE://
	CONFIRMSKIIS://
	CONFIRMBASE://
	LOWERSPA://
	CLAMPRETURN://
	CONFIRMSPAUNLOAD://
	
	
	
END_CASE
END_METHOD

METHOD homeMachine : BOOL
VAR_INPUT
END_VAR
homeMachine := FALSE;
CASE nHomeMachineState OF 
	0:// Home Motors
		IF aMoveFinish[2] THEN 
			IF NOT aMoveFinish[0] THEN
				(*CASE GVL_devices.fbLftClampMotor.homeToTorque() OF 
					1:// Done
						aMoveFinish[0] := TRUE;
					13:// Error
						GVL_devices.fbLftClampMotor.reset();
						GVL_machine.motorErrorList := LFTCLAMP;
						GVL_machine.bErrorPresent := TRUE;
				END_CASE*)
				IF GVL_devices.fbLftClampMotor.tempCylinderClose() THEN
					aMoveFinish[0] := TRUE;
				END_IF
			END_IF
		END_IF
		
		IF aMoveFinish[3] THEN
			IF NOT aMoveFinish[1] THEN
				CASE GVL_devices.fbRhtClampMotor.homeToTorque() OF 
					1:// Done
						aMoveFinish[1] := TRUE;
					13:// Error
						GVL_devices.fbRhtClampMotor.reset();
						GVL_machine.motorErrorList := RHTCLAMP;
						GVL_machine.bErrorPresent := TRUE;
				END_CASE
			END_IF
		END_IF
		
		IF NOT aMoveFinish[2] THEN
			CASE GVL_devices.fbLftWidthMotor.homeToSensorCustom() OF 
				1:// Done
					aMoveFinish[2] := TRUE;
				13:// Error
					GVL_machine.motorErrorList := LFTWIDTH;
					GVL_machine.bErrorPresent := TRUE;
			END_CASE
		END_IF
		IF NOT aMoveFinish[3] THEN
			CASE GVL_devices.fbRhtWidthMotor.homeToSensorCustom() OF 
				1:// Done
					aMoveFinish[3] := TRUE;
				13:// Error
					GVL_machine.motorErrorList := RHTWIDTH;
					GVL_machine.bErrorPresent := TRUE;
			END_CASE
		END_IF
		IF aMoveFinish[2] THEN
			IF NOT aMoveFinish[4] THEN
				CASE GVL_devices.fbLftRotationMotor.homeToTorque() OF 
					1:// Done
						aMoveFinish[4] := TRUE;
					13:// Error
						GVL_machine.motorErrorList := LFTROTATION;
						GVL_machine.bErrorPresent := TRUE;
				END_CASE
			END_IF
			IF NOT aMoveFinish[6] THEN
				IF GVL_devices.fbColumn1Motor.fbMotor.Status.Coupled THEN
					GVL_devices.fbColumn0Motor.motorIdle := FALSE;
					GVL_devices.fbColumn1Motor.motorIdle := FALSE;
					CASE GVL_devices.fbColumn0Motor.homeToSensor(0) OF 
						1:// Done
							aMoveFinish[6] := TRUE;
						13:// Error
							GVL_machine.motorErrorList := COLUMN0;
							GVL_machine.bErrorPresent := TRUE;
					END_CASE
				ELSE
					CASE GVL_devices.fbColumn1Motor.coupleToAxis(GVL_devices.fbColumn0Motor.fbMotor) OF 
						1:// Done
						13: GVL_devices.fbColumn1Motor.reset();
							GVL_machine.motorErrorList := COLUMN1;
							GVL_machine.bErrorPresent := TRUE;
					END_CASE
				END_IF
			END_IF
		END_IF
		
		IF aMoveFinish[3] THEN
			IF NOT aMoveFinish[5] THEN
				CASE GVL_devices.fbRhtRotationMotor.homeToTorque() OF 
					1:// Done
						aMoveFinish[5] := TRUE;
					13:// Error
						GVL_machine.motorErrorList := RHTROTATION;
						GVL_machine.bErrorPresent := TRUE;
				END_CASE
			END_IF
			
			IF NOT aMoveFinish[7] THEN
				IF GVL_devices.fbColumn3Motor.fbMotor.Status.Coupled THEN
					GVL_devices.fbColumn2Motor.motorIdle := FALSE;
					GVL_devices.fbColumn3Motor.motorIdle := FALSE;
					CASE GVL_devices.fbColumn2Motor.homeToSensor(0) OF 
						1:// Done
							aMoveFinish[7] := TRUE;
						13://Error
							GVL_machine.motorErrorList := COLUMN2;
							GVL_machine.bErrorPresent := TRUE;
					END_CASE
				ELSE
					CASE GVL_devices.fbColumn3Motor.coupleToAxis(GVL_devices.fbColumn2Motor.fbMotor) OF 
						1://Done 
						13: GVL_devices.fbColumn3Motor.reset();
							GVL_machine.motorErrorList := COLUMN3;
							GVL_machine.bErrorPresent := TRUE;
					END_CASE
				END_IF
			END_IF
		END_IF
			
		IF F_checkMoveFinish(aMoveFinish,8,FALSE) THEN
			nHomeMachineState := nHomeMachineState + 1;
		END_IF
	1:// Move rotation to 90 deg
		IF NOT aMoveFinish[0] THEN
			CASE GVL_devices.fbLftRotationMotor.moveTo('NULL',90/25.4) OF
				1: //Done
					aMoveFinish[0] := TRUE;
				13://Error
					GVL_machine.motorErrorList := LFTROTATION;
					GVL_machine.bErrorPresent := TRUE;
			END_CASE
		END_IF

		IF NOT aMoveFinish[1] THEN
			CASE GVL_devices.fbRhtRotationMotor.moveTo('NULL',90/25.4) OF
				1: //Done
					aMoveFinish[1] := TRUE;
				13://Error
					GVL_machine.motorErrorList := RHTROTATION;
					GVL_machine.bErrorPresent := TRUE;
			END_CASE
		END_IF	
		
		IF F_checkMoveFinish(aMoveFinish,2,FALSE) THEN
			nHomeMachineState := nHomeMachineState + 1;
		END_IF
		
	2:// Decouple all Motors
		IF NOT GVL_devices.fbColumn1Motor.fbMotor.Status.Coupled AND NOT GVL_devices.fbColumn3Motor.fbMotor.Status.Coupled THEN
			aMoveFinish[0] := TRUE;
		ELSE
			GVL_devices.fbColumn1Motor.decoupleAxis();
			GVL_devices.fbColumn3Motor.decoupleAxis();
		END_IF
		
		
		// Set Slave motors to same counts as their masters after homing sequence
		IF aMoveFinish[0] THEN
			IF NOT aMoveFinish[1] THEN
				CASE GVL_devices.fbColumn1Motor.homeSetToCount(GVL_devices.fbColumn0Motor.fbMotor.NcToPlc.ActPos) OF
					1:// Done
						aMoveFinish[1] := TRUE;
					13:// Error
						GVL_machine.motorErrorList := COLUMN1;
						GVL_machine.bErrorPresent := TRUE;
				END_CASE
			END_IF
			IF NOT aMoveFinish[2] THEN
				CASE GVL_devices.fbColumn3Motor.homeSetToCount(GVL_devices.fbColumn2Motor.fbMotor.NcToPlc.ActPos) OF
					1:// Done
						aMoveFinish[2] := TRUE;
					13:// Error
						GVL_machine.motorErrorList := COLUMN3;
						GVL_machine.bErrorPresent := TRUE;
				END_CASE
			END_IF
		END_IF
		
		IF F_checkMoveFinish(aMoveFinish,3,FALSE) THEN
			nHomeMachineState := 0;
			homeMachine := TRUE;
		END_IF
END_CASE
END_METHOD

METHOD motorFault : BOOL
VAR_INPUT
END_VAR
motorFault := FALSE;
IF GVL_devices.fbColumn0Motor.fbMotor.Status.Error OR
	GVL_devices.fbColumn1Motor.fbMotor.Status.Error OR
	GVL_devices.fbColumn2Motor.fbMotor.Status.Error OR
	GVL_devices.fbColumn3Motor.fbMotor.Status.Error OR
	GVL_devices.fbLftClampMotor.fbMotor.Status.Error OR
	GVL_devices.fbRhtClampMotor.fbMotor.Status.Error OR
	GVL_devices.fbLftWidthMotor.fbMotor.Status.Error OR
	GVL_devices.fbRhtWidthMotor.fbMotor.Status.Error OR
	GVL_devices.fbLftRotationMotor.fbMotor.Status.Error OR
	GVL_devices.fbRhtRotationMotor.fbMotor.Status.Error THEN
	motorFault := TRUE;
END_IF
END_METHOD

METHOD moveColumns : INT
VAR_INPUT
	sState : STRING;
	fHeight : REAL;
	nOption : INT; //0 - Left Columns and Right Columns Move Seperate, 1- All columns follow one Master
END_VAR
moveColumns := 0;
CASE nOption OF 
	0:// Left Columns and Right Columns Move Seperate
		
	1:// All columns follow one Master
		CASE nMoveColumnState OF 
			0: // Execute Move on Master Axis 
				IF GVL_devices.fbColumn1Motor.fbMotor.Status.Coupled AND GVL_devices.fbColumn2Motor.fbMotor.Status.Coupled AND GVL_devices.fbColumn3Motor.fbMotor.Status.Coupled THEN
					GVL_devices.fbColumn0Motor.motorIdle := FALSE;
					GVL_devices.fbColumn1Motor.motorIdle := FALSE;
					GVL_devices.fbColumn2Motor.motorIdle := FALSE;
					GVL_devices.fbColumn3Motor.motorIdle := FALSE;
					CASE GVL_devices.fbColumn0Motor.moveTo(sState,fHeight) OF 
						1: //Done
							nMoveColumnState := nMoveColumnState + 1;
						13: //Error
							GVL_machine.motorErrorList := COLUMN0;
							GVL_machine.bErrorPresent := TRUE;
							moveColumns := 13;
						15: //Move is halfway
							moveColumns := 15;
					END_CASE
					IF GVL_devices.fbColumn0Motor.fbMotor.Status.Error OR GVL_devices.fbColumn1Motor.fbMotor.Status.Error OR GVL_devices.fbColumn2Motor.fbMotor.Status.Error OR GVL_devices.fbColumn3Motor.fbMotor.Status.Error THEN
						GVL_devices.fbColumn0Motor.estop();
						GVL_devices.fbColumn1Motor.estop();
						GVL_devices.fbColumn2Motor.estop();
						GVL_devices.fbColumn3Motor.estop();
						moveColumns := 13;
					END_IF
				ELSE
					CASE GVL_devices.fbColumn1Motor.coupleToAxis(GVL_devices.fbColumn0Motor.fbMotor) OF
						1:// Done
						13:// Error
							GVL_machine.motorErrorList := COLUMN1;
							GVL_machine.bErrorPresent := TRUE;
					END_CASE
					CASE GVL_devices.fbColumn2Motor.coupleToAxis(GVL_devices.fbColumn0Motor.fbMotor) OF
						1:// Done
						13:// Error
							GVL_machine.motorErrorList := COLUMN2;
							GVL_machine.bErrorPresent := TRUE;
					END_CASE
					CASE GVL_devices.fbColumn3Motor.coupleToAxis(GVL_devices.fbColumn0Motor.fbMotor) OF
						1:// Done
						13:// Error
							GVL_machine.motorErrorList := COLUMN3;
							GVL_machine.bErrorPresent := TRUE;
					END_CASE
				END_IF
			1:// Decouple Axis
				IF NOT GVL_devices.fbColumn1Motor.fbMotor.Status.Coupled AND NOT GVL_devices.fbColumn2Motor.fbMotor.Status.Coupled AND NOT GVL_devices.fbColumn3Motor.fbMotor.Status.Coupled THEN
					nMoveColumnState := 0;
					moveColumns := 1;
				ELSE
					GVL_devices.fbColumn1Motor.decoupleAxis();
					GVL_devices.fbColumn2Motor.decoupleAxis();
					GVL_devices.fbColumn3Motor.decoupleAxis();
				END_IF
		END_CASE
END_CASE
END_METHOD

METHOD moveRotation : INT
VAR_INPUT
	sState : STRING;
	fHeight : REAL;
END_VAR
moveRotation := 0;
CASE nMoveRotationState OF 
	0://Command Move
		IF NOT aMoveFinishSecond[0] THEN
			CASE GVL_devices.fbLftRotationMotor.moveTo(sState,fHeight/25.4) OF 
				1:// Done
					aMoveFinishSecond[0] := TRUE;
				13:// Errror
					GVL_machine.motorErrorList := LFTROTATION;
					GVL_machine.bErrorPresent := TRUE;
					moveRotation := 13;
			END_CASE
		END_IF
		IF NOT aMoveFinishSecond[1] THEN
			CASE GVL_devices.fbRhtRotationMotor.moveTo(sState,fHeight/25.4) OF
				1:// Done
					aMoveFinishSecond[1] := TRUE;
				13:// Error
					GVL_machine.motorErrorList := RHTROTATION;
					GVL_machine.bErrorPresent := TRUE;
					moveRotation := 13;
				15:// Move halfway
					moveRotation := 15;
			END_CASE
		END_IF
		
		//Check if move is finished
		IF F_checkMoveFinish(aMoveFinishSecond,2,FALSE) THEN
			moveRotation := 1;
		END_IF
		
		//Check if one is moving without other
		IF GVL_devices.fbLftRotationMotor.fbMotor.Status.Moving OR GVL_devices.fbRhtRotationMotor.fbMotor.Status.Moving THEN
			IF GVL_devices.fbLftRotationMotor.fbMotor.Status.NotMoving OR GVL_devices.fbRhtRotationMotor.fbMotor.Status.NotMoving THEN
				fbMoveDelayTimRot(IN := TRUE, PT := T#500MS);
				IF fbMoveDelayTimRot.Q THEN
					moveRotation := 13;
				END_IF
			ELSE
				fbMoveDelayTimRot(IN := FALSE);
			END_IF
		END_IF
		
		(*IF GVL_devices.fbLftRotationMotor.fbMotor.Status.Moving AND NOT GVL_devices.fbRhtRotationMotor.fbMotor.Status.Moving THEN
			moveRotation := 13;
		ELSIF NOT GVL_devices.fbLftRotationMotor.fbMotor.Status.Moving AND GVL_devices.fbRhtRotationMotor.fbMotor.Status.Moving THEN
			moveRotation := 13;
		END_IF*)
END_CASE
END_METHOD

METHOD resetAutoProgram : INT
VAR_INPUT
END_VAR
CASE eResetState OF 
	CHECKWIDTH:
		sPromptDisp := 'RESET: Checking Width';
		F_checkMoveFinish(aMoveFinish,0,TRUE);
		IF GVL_devices.fbLftWidthMotor.distance < 1  AND GVL_devices.fbRhtWidthMotor.distance < 1 THEN
			eResetState := RESETDONE;
		ELSE
			eResetState := CHECKCLAMPS;
		END_IF
	
	CHECKCLAMPS:
		sPromptDisp := 'RESET: Checking Clamps';
		IF (GVL_devices.fbLftClampMotor.distance > -1 AND GVL_devices.fbRhtClampMotor.distance < 1) OR (GVL_devices.fbLftClampMotor.distance < -130 AND GVL_devices.fbRhtClampMotor.distance > 130) THEN
			eResetState := RESETDONE;
		ELSE
			eResetState := CHECKROTATION;
		END_IF
		
	CHECKROTATION:
		sPromptDisp := 'RESET: Checking Rotation';
		IF GVL_devices.fbLftRotationMotor.distance = -90 AND GVL_devices.fbRhtRotationMotor.distance = 90 THEN
			eResetState := CHECKHEIGHT;
		ELSIF GVL_devices.fbLftRotationMotor.distance = -270 AND GVL_devices.fbRhtRotationMotor.distance = 270 THEN
			eResetState := MOVETOFLIPHEIGHT;
		ELSE
			eResetState := MOVETOFLIPHEIGHT;
		END_IF
		
	CHECKHEIGHT://Check Height of Columns
		sPromptDisp := 'RESET: Checking Columns';
		IF GVL_devices.fbColumn0Motor.distance > -1 THEN
			eResetState := OPENCLAMPS;
		ELSE
			sPromptDisp := 'RESET: Moving Columns';
			CASE moveColumns('NULL',0,1) OF 
				1: // Done
					eResetState := OPENCLAMPS;
				13:// error 
					GVL_devices.fbColumn0Motor.stop();
					GVL_devices.fbColumn1Motor.stop();
					GVL_devices.fbColumn2Motor.stop();
					GVL_devices.fbColumn3Motor.stop();
					ePrevState := RESETPROGRAM;
					eState := PROGERRORSTOP;
					sPromptDisp := 'Column Faulted Retry Start';
			END_CASE
		END_IF
		
	MOVETOFLIPHEIGHT: //Move Spa to eflex flip height and unwind rotation. 
		sPromptDisp := 'RESET: Rotating Spa';
			IF NOT aMoveFinish[0] THEN
				IF GVL_eflex.fFlipHeight > 12 THEN
					CASE moveColumns('NULL',GVL_eflex.fFlipHeight,1) OF 
						1:// Done
							aMoveFinish[0] := TRUE;
							aMoveFinish[1] := TRUE;
						13:// Error
							GVL_devices.fbColumn0Motor.stop();
							GVL_devices.fbColumn1Motor.stop();
							GVL_devices.fbColumn2Motor.stop();
							GVL_devices.fbColumn3Motor.stop();
							ePrevState := RESETPROGRAM;
							eState := PROGERRORSTOP;
							sPromptDisp := 'Column Faulted Retry Start';
						15:// Move is halway
							aMoveFinish[1] := TRUE;
					END_CASE
				ELSE
					CASE moveColumns('NULL',24,1) OF 
						1:// Done
							aMoveFinish[0] := TRUE;
						13:// Error
							GVL_devices.fbColumn0Motor.stop();
							GVL_devices.fbColumn1Motor.stop();
							GVL_devices.fbColumn2Motor.stop();
							GVL_devices.fbColumn3Motor.stop();
							ePrevState := RESETPROGRAM;
							eState := PROGERRORSTOP;
							sPromptDisp := 'Column Faulted Retry Start';
						15:// Move is halway
							aMoveFinish[1] := TRUE;
					END_CASE
				END_IF
			END_IF
			IF aMoveFinish[1] THEN
				IF NOT aMoveFinish[2] THEN
					CASE moveRotation('NULL',90) OF 
						1:// Done
							aMoveFinish[2] := TRUE;
						13:// Error
							GVL_devices.fbLftRotationMotor.stop();
							GVL_devices.fbRhtRotationMotor.stop();
						15:// Move Halfway	
							aMoveFinish[3] := TRUE;
					END_CASE
				END_IF
			END_IF
			
			IF NOT aMoveFinish[4] THEN
				IF GVL_devices.fbTable.moveTo(GVL_persistent.fTableDownHeight) THEN
					aMoveFinish[4] := TRUE;
				END_IF
			END_IF
		
			IF F_checkMoveFinish(aMoveFinish,5,FALSE) THEN
				eResetState := MOVETOUNCLAMPHEIGHT;
			END_IF

	MOVETOUNCLAMPHEIGHT:
		sPromptDisp := 'RESET: Releasing Spa';
		IF NOT aMoveFinish[0] THEN
			CASE moveColumns('NULL',0,1) OF 
				1:// Done
					aMoveFinish[0] := TRUE;
				13:// Error
					GVL_devices.fbColumn0Motor.stop();
					GVL_devices.fbColumn1Motor.stop();
					GVL_devices.fbColumn2Motor.stop();
					GVL_devices.fbColumn3Motor.stop();
					ePrevState := RESETPROGRAM;
					eState := PROGERRORSTOP;
					sPromptDisp := 'Column Faulted Retry Start';
				15:// Move is halway
					aMoveFinish[1] := TRUE;
			END_CASE
		END_IF
		
		IF aMoveFinish[1] THEN
			IF NOT aMoveFinish[2] THEN
				CASE GVL_devices.fbLftClampMotor.moveTo('NULL',GVL_persistent.fClampOpenDist) OF 
					1: // Done
						aMoveFinish[2] := TRUE;
					13://pass
				END_CASE
			END_IF
			IF NOT aMoveFinish[3] THEN
				CASE GVL_devices.fbRhtClampMotor.moveTo('NULL',GVL_persistent.fClampOpenDist) OF 
					1: // Done
						aMoveFinish[3] := TRUE;
					13://pass
				END_CASE
			END_IF
			IF NOT aMoveFinish[4] THEN
				IF GVL_devices.fbTable.moveTo(GVL_persistent.fTableClampHeight) THEN
					aMoveFinish[4] := TRUE;
				END_IF
			END_IF
		END_IF
		
		IF F_checkMoveFinish(aMoveFinish,5,FALSE) THEN
			eResetState := RESETDONE;
		END_IF
		
	OPENCLAMPS://pass
		sPromptDisp := 'RESET: Opening Clamps';
		IF NOT aMoveFinish[0] THEN
			IF GVL_devices.fbTable.moveTo(GVL_persistent.fTableClampHeight) THEN
				aMoveFinish[0] := TRUE;
			END_IF
		END_IF
		
		IF NOT aMoveFinish[1] THEN
			CASE GVL_devices.fbLftClampMotor.moveTo('NULL',GVL_persistent.fClampOpenDist) OF 
				1: // Done
					aMoveFinish[1] := TRUE;
				13://pass
			END_CASE
		END_IF
		IF NOT aMoveFinish[2] THEN
			CASE GVL_devices.fbRhtClampMotor.moveTo('NULL',GVL_persistent.fClampOpenDist) OF 
				1: // Done
					aMoveFinish[2] := TRUE;
				13://pass
			END_CASE
		END_IF
		
		IF F_checkMoveFinish(aMoveFinish,4,FALSE) THEN
			eResetState := RESETDONE;
		END_IF
		
	RESETDONE:// SteadyState
		sPromptDisp := 'RESET: Reset Done';
END_CASE
END_METHOD

END_PROGRAM

// ---- POUs/FUNCTIONS/F_checkMoveFinish.TcPOU
FUNCTION F_checkMoveFinish : BOOL
VAR_INPUT
	refArray 	: REFERENCE TO ARRAY[0..10] OF BOOL; //Move finish array to check 
	nCount		: INT; // Number of moves completed to check against
	reset		: BOOL; // True - Resets array, False - checks array against nCount;
END_VAR
VAR
	nCounter 	: INT := 0;
	i 			: INT := 0;
END_VAR

F_checkMoveFinish := FALSE;
IF NOT reset THEN 
	FOR i := 0 TO SIZEOF(refArray)-1 BY 1 DO
		IF refArray[i] THEN 
			nCounter := nCounter + 1;
		END_IF
	END_FOR
	
